{attribute 'qualified_only'}
{attribute 'global_init_slot' := '50500'}
VAR_GLOBAL PERSISTENT
	//These tags are created here because you cannot write directly to local scoped tags(cpt_3144) from outside the POU
	//They are created here then mapped to the local variables in the POU
	//All tags in this GVL MUST have the {attribute 'OPC.UA.DA' :='1'} string above them in order to be exposed to OPC
	//Tags that are ONLY being read from the HMI have their values set in the opc_mapping program
	
	//------------------------------------------------------------------------------------------------------------------


	//---System date time year-----------------------------------------------------------------------------------------------
	{attribute 'OPC.UA.DA' :='1'}
	popa_0082_system_date_time_year : INT;
	//System date time month
	{attribute 'OPC.UA.DA' :='1'}
	popa_0082_system_date_time_month : INT;
	//System date time day
	{attribute 'OPC.UA.DA' :='1'}
	popa_0082_system_date_time_day : INT;
	//System date time hour
	{attribute 'OPC.UA.DA' :='1'}
	popa_0082_system_date_time_hour : INT;
	//System date time minute
	{attribute 'OPC.UA.DA' :='1'}
	popa_0082_system_date_time_minute : INT;
	//System date time second
	{attribute 'OPC.UA.DA' :='1'}
	popa_0082_system_date_time_second : INT;
	//Hour setpoint for daily reset triggers
	{attribute 'OPC.UA.DA' :='1'}
	popa_0082_daily_reset_hour_setpoint : INT;
	//Minute setpoint for daily reset triggers
	{attribute 'OPC.UA.DA' :='1'}
	popa_0082_daily_reset_minute_setpoint : INT;
	//Alarm acknowledge, acks all alarms, clears lower priority level alarms
	{attribute 'OPC.UA.DA' :='1'}
	popa_0082_alarm_ack : BOOL;
	//Alarm reset, clears higher priority alarms
	{attribute 'OPC.UA.DA' :='1'}
	popa_0082_alarm_reset : BOOL;
	
//----------------------------------------------------------------------------------------------------------------------------------------		
	//State Mode
	{attribute 'OPC.UA.DA' :='1'}
	popa_0082_ed_routine_maint : BOOL;
	{attribute 'OPC.UA.DA' :='1'}
	popa_0082_ed_routine_idle : BOOL;
	{attribute 'OPC.UA.DA' :='1'}
	popa_0082_ed_routine_cip : BOOL;
	{attribute 'OPC.UA.DA' :='1'}
	popa_0082_ed_routine_stop : BOOL;
	{attribute 'OPC.UA.DA' :='1'}
	popa_0082_ed_routine_critical_stop : BOOL;
	
	
	//Safety
	{attribute 'OPC.UA.DA' :='1'}
	popa_0082_ed_safety_reset : BOOL;
	
	
//---HMI Commands--------------------------------------------------------------------------------------------------------------------------------------

	//Setpoints------------------------------------------------------------------------------------------------------------------
	{attribute 'OPC.UA.DA' :='1'}
	popa_0082_idle_pressure_setpoint_request : REAL;
	{attribute 'OPC.UA.DA' :='1'}
	popa_0082_cip_pressure_setpoint_request : REAL;
	{attribute 'OPC.UA.DA' :='1'}
	popa_0082_av_3148_b_hmi_position_request : REAL;
	{attribute 'OPC.UA.DA' :='1'}
	popa_0082_av_3248_b_hmi_position_request : REAL;
	{attribute 'OPC.UA.DA' :='1'}
	popa_0082_av_3348_b_hmi_position_request : REAL;
	
	//Pumps-----------------------------------------------------------------------------------------------------------------------
	{attribute 'OPC.UA.DA' :='1'}
	popa_0082_u_3112_b_hmi_start_request: BOOL;
	{attribute 'OPC.UA.DA' :='1'}
	popa_0082_u_3212_b_hmi_start_request: BOOL;
	{attribute 'OPC.UA.DA' :='1'}
	popa_0082_u_3312_b_hmi_start_request: BOOL;
	{attribute 'OPC.UA.DA' :='1'}
	popa_0082_u_3160_b_hmi_start_request: BOOL;
	{attribute 'OPC.UA.DA' :='1'}
	popa_0082_u_3260_b_hmi_start_request: BOOL;
	{attribute 'OPC.UA.DA' :='1'}
	popa_0082_u_3360_b_hmi_start_request: BOOL;
	{attribute 'OPC.UA.DA' :='1'}
	popa_0082_u_3370_b_hmi_start_request: BOOL;
	{attribute 'OPC.UA.DA' :='1'}
	popa_0092_u_3405_b_hmi_start_request: BOOL;
		
	{attribute 'OPC.UA.DA' :='1'}
	popa_0082_u_3112_b_hmi_speed_request: REAL;
	{attribute 'OPC.UA.DA' :='1'}
	popa_0082_u_3212_b_hmi_speed_request: REAL;
	{attribute 'OPC.UA.DA' :='1'}
	popa_0082_u_3312_b_hmi_speed_request: REAL;
	{attribute 'OPC.UA.DA' :='1'}
	popa_0082_u_3160_b_hmi_speed_request: REAL;
	{attribute 'OPC.UA.DA' :='1'}
	popa_0082_u_3260_b_hmi_speed_request: REAL;
	{attribute 'OPC.UA.DA' :='1'}
	popa_0082_u_3360_b_hmi_speed_request: REAL;
	{attribute 'OPC.UA.DA' :='1'}
	popa_0082_u_3370_b_hmi_speed_request: REAL;
	{attribute 'OPC.UA.DA' :='1'}
	popa_0092_u_3405_b_hmi_speed_request: REAL;
	
	//Valves------------------------------------------------------------------------------------------------------------------------------
	{attribute 'OPC.UA.DA' :='1'}
	popa_0082_nv_3110_b_hmi_open_request: BOOL;
	{attribute 'OPC.UA.DA' :='1'}
	popa_0082_nv_3210_b_hmi_open_request: BOOL;
	{attribute 'OPC.UA.DA' :='1'}
	popa_0082_nv_3310_b_hmi_open_request: BOOL;
	{attribute 'OPC.UA.DA' :='1'}
	popa_0082_nv_3135_b_hmi_open_request: BOOL;
	{attribute 'OPC.UA.DA' :='1'}
	popa_0082_nv_3235_b_hmi_open_request: BOOL;
	{attribute 'OPC.UA.DA' :='1'}
	popa_0082_nv_3335_b_hmi_open_request: BOOL;
	{attribute 'OPC.UA.DA' :='1'}
	popa_0082_nv_3372_b_hmi_open_request: BOOL;
	{attribute 'OPC.UA.DA' :='1'}
	popa_0082_nv_3162_b_hmi_open_request: BOOL;
	

	//-------------------------------------------------------------------------------------------
	//Digital valve open request
	{attribute 'OPC.UA.DA' :='1'}
	popa_0082_nv_3110_b_open_request : BOOL;
	//Digital valve status
	{attribute 'OPC.UA.DA' :='1'}
	popa_0082_nv_3110_b_status : INT;
	
	//Digital valve open request
	{attribute 'OPC.UA.DA' :='1'}
	popa_0082_nv_3210_b_open_request : BOOL;
	//Digital valve status
	{attribute 'OPC.UA.DA' :='1'}
	popa_0082_nv_3210_b_status : INT;
	
	//Digital valve open request
	{attribute 'OPC.UA.DA' :='1'}
	popa_0082_nv_3310_b_open_request : BOOL;
	//Digital valve status
	{attribute 'OPC.UA.DA' :='1'}
	popa_0082_nv_3310_b_status : INT;
	
	//Digital valve open request
	{attribute 'OPC.UA.DA' :='1'}
	popa_0082_nv_3135_b_open_request : BOOL;
	//Digital valve status
	{attribute 'OPC.UA.DA' :='1'}
	popa_0082_nv_3135_b_status : INT;
	
	//Digital valve open request
	{attribute 'OPC.UA.DA' :='1'}
	popa_0082_nv_3235_b_open_request : BOOL;
	//Digital valve status
	{attribute 'OPC.UA.DA' :='1'}
	popa_0082_nv_3235_b_status : INT;
	
	//Digital valve open request
	{attribute 'OPC.UA.DA' :='1'}
	popa_0082_nv_3335_b_open_request : BOOL;
	//Digital valve status
	{attribute 'OPC.UA.DA' :='1'}
	popa_0082_nv_3335_b_status : INT;
	
	//Digital valve open request
	{attribute 'OPC.UA.DA' :='1'}
	popa_0082_nv_3372_b_open_request : BOOL;
	//Digital valve status
	{attribute 'OPC.UA.DA' :='1'}
	popa_0082_nv_3372_b_status : INT;
	
	//Digital valve open request
	{attribute 'OPC.UA.DA' :='1'}
	popa_0082_nv_3162_b_open_request : BOOL;
	//Digital valve status
	{attribute 'OPC.UA.DA' :='1'}
	popa_0082_nv_3162_b_status : INT;
	
	//------------------------------------------------------------------------------------------------------------------
	//Alarm Priority setpoint
	{attribute 'OPC.UA.DA' :='1'}
	popa_0082_av_3148_b_position_fail_priority : INT;
	//Alarm delay setpoint(seconds)
	{attribute 'OPC.UA.DA' :='1'}
	popa_0082_av_3148_b_position_fail_delay_setpoint : INT;
	//Alarm active for HMI
	{attribute 'OPC.UA.DA' :='1'}
	popa_0082_av_3148_b_position_fail_active : BOOL;
	//Alarm enable
	{attribute 'OPC.UA.DA' :='1'}
	popa_0082_av_3148_b_position_fail_enable: BOOL;
	//------------------------------------------------------------------------------------------------------------------
	//Alarm Priority setpoint
	{attribute 'OPC.UA.DA' :='1'}
	popa_0082_av_3248_b_position_fail_priority : INT;
	//Alarm delay setpoint(seconds)
	{attribute 'OPC.UA.DA' :='1'}
	popa_0082_av_3248_b_position_fail_delay_setpoint : INT;
	//Alarm active for HMI
	{attribute 'OPC.UA.DA' :='1'}
	popa_0082_av_3248_b_position_fail_active : BOOL;
	//Alarm enable
	{attribute 'OPC.UA.DA' :='1'}
	popa_0082_av_3248_b_position_fail_enable: BOOL;
	//------------------------------------------------------------------------------------------------------------------
	//Alarm Priority setpoint
	{attribute 'OPC.UA.DA' :='1'}
	popa_0082_av_3348_b_position_fail_priority : INT;
	//Alarm delay setpoint(seconds)
	{attribute 'OPC.UA.DA' :='1'}
	popa_0082_av_3348_b_position_fail_delay_setpoint : INT;
	//Alarm active for HMI
	{attribute 'OPC.UA.DA' :='1'}
	popa_0082_av_3348_b_position_fail_active : BOOL;
	//Alarm enable
	{attribute 'OPC.UA.DA' :='1'}
	popa_0082_av_3348_b_position_fail_enable: BOOL;
	
	//------------------------------------------------------------------------------------------------------------------
	//Alarm Priority setpoint
	{attribute 'OPC.UA.DA' :='1'}
	popa_0082_nv_3110_b_fail_to_open_priority : INT;
	//Alarm delay setpoint(seconds)
	{attribute 'OPC.UA.DA' :='1'}
	popa_0082_nv_3110_b_fail_to_open_delay_setpoint : INT;
	//Alarm active for HMI
	{attribute 'OPC.UA.DA' :='1'}
	popa_0082_nv_3110_b_fail_to_open_active : BOOL;
	//Alarm enable
	{attribute 'OPC.UA.DA' :='1'}
	popa_0082_nv_3110_b_fail_to_open_enable: BOOL;
	
	//Alarm Priority setpoint
	{attribute 'OPC.UA.DA' :='1'}
	popa_0082_nv_3110_b_fail_to_close_priority : INT;
	//Alarm delay setpoint(seconds)
	{attribute 'OPC.UA.DA' :='1'}
	popa_0082_nv_3110_b_fail_to_close_delay_setpoint : INT;
	//Alarm active for HMI
	{attribute 'OPC.UA.DA' :='1'}
	popa_0082_nv_3110_b_fail_to_close_active : BOOL;
	//Alarm enable
	{attribute 'OPC.UA.DA' :='1'}
	popa_0082_nv_3110_b_fail_to_close_enable: BOOL;
	
	//------------------------------------------------------------------------------------------------------------------
	//Alarm Priority setpoint
	{attribute 'OPC.UA.DA' :='1'}
	popa_0082_nv_3210_b_fail_to_open_priority : INT;
	//Alarm delay setpoint(seconds)
	{attribute 'OPC.UA.DA' :='1'}
	popa_0082_nv_3210_b_fail_to_open_delay_setpoint : INT;
	//Alarm active for HMI
	{attribute 'OPC.UA.DA' :='1'}
	popa_0082_nv_3210_b_fail_to_open_active : BOOL;
	//Alarm enable
	{attribute 'OPC.UA.DA' :='1'}
	popa_0082_nv_3210_b_fail_to_open_enable: BOOL;
	
	//Alarm Priority setpoint
	{attribute 'OPC.UA.DA' :='1'}
	popa_0082_nv_3210_b_fail_to_close_priority : INT;
	//Alarm delay setpoint(seconds)
	{attribute 'OPC.UA.DA' :='1'}
	popa_0082_nv_3210_b_fail_to_close_delay_setpoint : INT;
	//Alarm active for HMI
	{attribute 'OPC.UA.DA' :='1'}
	popa_0082_nv_3210_b_fail_to_close_active : BOOL;
	//Alarm enable
	{attribute 'OPC.UA.DA' :='1'}
	popa_0082_nv_3210_b_fail_to_close_enable: BOOL;
	
	//------------------------------------------------------------------------------------------------------------------
	//Alarm Priority setpoint
	{attribute 'OPC.UA.DA' :='1'}
	popa_0082_nv_3310_b_fail_to_open_priority : INT;
	//Alarm delay setpoint(seconds)
	{attribute 'OPC.UA.DA' :='1'}
	popa_0082_nv_3310_b_fail_to_open_delay_setpoint : INT;
	//Alarm active for HMI
	{attribute 'OPC.UA.DA' :='1'}
	popa_0082_nv_3310_b_fail_to_open_active : BOOL;
	//Alarm enable
	{attribute 'OPC.UA.DA' :='1'}
	popa_0082_nv_3310_b_fail_to_open_enable: BOOL;
	
	//Alarm Priority setpoint
	{attribute 'OPC.UA.DA' :='1'}
	popa_0082_nv_3310_b_fail_to_close_priority : INT;
	//Alarm delay setpoint(seconds)
	{attribute 'OPC.UA.DA' :='1'}
	popa_0082_nv_3310_b_fail_to_close_delay_setpoint : INT;
	//Alarm active for HMI
	{attribute 'OPC.UA.DA' :='1'}
	popa_0082_nv_3310_b_fail_to_close_active : BOOL;
	//Alarm enable
	{attribute 'OPC.UA.DA' :='1'}
	popa_0082_nv_3310_b_fail_to_close_enable: BOOL;
	
	//------------------------------------------------------------------------------------------------------------------
	//Alarm Priority setpoint
	{attribute 'OPC.UA.DA' :='1'}
	popa_0082_nv_3135_b_fail_to_open_priority : INT;
	//Alarm delay setpoint(seconds)
	{attribute 'OPC.UA.DA' :='1'}
	popa_0082_nv_3135_b_fail_to_open_delay_setpoint : INT;
	//Alarm active for HMI
	{attribute 'OPC.UA.DA' :='1'}
	popa_0082_nv_3135_b_fail_to_open_active : BOOL;
	//Alarm enable
	{attribute 'OPC.UA.DA' :='1'}
	popa_0082_nv_3135_b_fail_to_open_enable: BOOL;
	
	//Alarm Priority setpoint
	{attribute 'OPC.UA.DA' :='1'}
	popa_0082_nv_3135_b_fail_to_close_priority : INT;
	//Alarm delay setpoint(seconds)
	{attribute 'OPC.UA.DA' :='1'}
	popa_0082_nv_3135_b_fail_to_close_delay_setpoint : INT;
	//Alarm active for HMI
	{attribute 'OPC.UA.DA' :='1'}
	popa_0082_nv_3135_b_fail_to_close_active : BOOL;
	//Alarm enable
	{attribute 'OPC.UA.DA' :='1'}
	popa_0082_nv_3135_b_fail_to_close_enable: BOOL;
	
	//------------------------------------------------------------------------------------------------------------------
	//Alarm Priority setpoint
	{attribute 'OPC.UA.DA' :='1'}
	popa_0082_nv_3235_b_fail_to_open_priority : INT;
	//Alarm delay setpoint(seconds)
	{attribute 'OPC.UA.DA' :='1'}
	popa_0082_nv_3235_b_fail_to_open_delay_setpoint : INT;
	//Alarm active for HMI
	{attribute 'OPC.UA.DA' :='1'}
	popa_0082_nv_3235_b_fail_to_open_active : BOOL;
	//Alarm enable
	{attribute 'OPC.UA.DA' :='1'}
	popa_0082_nv_3235_b_fail_to_open_enable: BOOL;
	
	//Alarm Priority setpoint
	{attribute 'OPC.UA.DA' :='1'}
	popa_0082_nv_3235_b_fail_to_close_priority : INT;
	//Alarm delay setpoint(seconds)
	{attribute 'OPC.UA.DA' :='1'}
	popa_0082_nv_3235_b_fail_to_close_delay_setpoint : INT;
	//Alarm active for HMI
	{attribute 'OPC.UA.DA' :='1'}
	popa_0082_nv_3235_b_fail_to_close_active : BOOL;
	//Alarm enable
	{attribute 'OPC.UA.DA' :='1'}
	popa_0082_nv_3235_b_fail_to_close_enable: BOOL;
	
	//------------------------------------------------------------------------------------------------------------------
	//Alarm Priority setpoint
	{attribute 'OPC.UA.DA' :='1'}
	popa_0082_nv_3335_b_fail_to_open_priority : INT;
	//Alarm delay setpoint(seconds)
	{attribute 'OPC.UA.DA' :='1'}
	popa_0082_nv_3335_b_fail_to_open_delay_setpoint : INT;
	//Alarm active for HMI
	{attribute 'OPC.UA.DA' :='1'}
	popa_0082_nv_3335_b_fail_to_open_active : BOOL;
	//Alarm enable
	{attribute 'OPC.UA.DA' :='1'}
	popa_0082_nv_3335_b_fail_to_open_enable: BOOL;
	
	//Alarm Priority setpoint
	{attribute 'OPC.UA.DA' :='1'}
	popa_0082_nv_3335_b_fail_to_close_priority : INT;
	//Alarm delay setpoint(seconds)
	{attribute 'OPC.UA.DA' :='1'}
	popa_0082_nv_3335_b_fail_to_close_delay_setpoint : INT;
	//Alarm active for HMI
	{attribute 'OPC.UA.DA' :='1'}
	popa_0082_nv_3335_b_fail_to_close_active : BOOL;
	//Alarm enable
	{attribute 'OPC.UA.DA' :='1'}
	popa_0082_nv_3335_b_fail_to_close_enable: BOOL;
	
	//------------------------------------------------------------------------------------------------------------------
	//Alarm Priority setpoint
	{attribute 'OPC.UA.DA' :='1'}
	popa_0082_nv_3372_b_fail_to_open_priority : INT;
	//Alarm delay setpoint(seconds)
	{attribute 'OPC.UA.DA' :='1'}
	popa_0082_nv_3372_b_fail_to_open_delay_setpoint : INT;
	//Alarm active for HMI
	{attribute 'OPC.UA.DA' :='1'}
	popa_0082_nv_3372_b_fail_to_open_active : BOOL;
	//Alarm enable
	{attribute 'OPC.UA.DA' :='1'}
	popa_0082_nv_3372_b_fail_to_open_enable: BOOL;
	
	//Alarm Priority setpoint
	{attribute 'OPC.UA.DA' :='1'}
	popa_0082_nv_3372_b_fail_to_close_priority : INT;
	//Alarm delay setpoint(seconds)
	{attribute 'OPC.UA.DA' :='1'}
	popa_0082_nv_3372_b_fail_to_close_delay_setpoint : INT;
	//Alarm active for HMI
	{attribute 'OPC.UA.DA' :='1'}
	popa_0082_nv_3372_b_fail_to_close_active : BOOL;
	//Alarm enable
	{attribute 'OPC.UA.DA' :='1'}
	popa_0082_nv_3372_b_fail_to_close_enable: BOOL;
	
	//------------------------------------------------------------------------------------------------------------------
	//Alarm Priority setpoint
	{attribute 'OPC.UA.DA' :='1'}
	popa_0082_nv_3162_b_fail_to_open_priority : INT;
	//Alarm delay setpoint(seconds)
	{attribute 'OPC.UA.DA' :='1'}
	popa_0082_nv_3162_b_fail_to_open_delay_setpoint : INT;
	//Alarm active for HMI
	{attribute 'OPC.UA.DA' :='1'}
	popa_0082_nv_3162_b_fail_to_open_active : BOOL;
	//Alarm enable
	{attribute 'OPC.UA.DA' :='1'}
	popa_0082_nv_3162_b_fail_to_open_enable: BOOL;
	
	//Alarm Priority setpoint
	{attribute 'OPC.UA.DA' :='1'}
	popa_0082_nv_3162_b_fail_to_close_priority : INT;
	//Alarm delay setpoint(seconds)
	{attribute 'OPC.UA.DA' :='1'}
	popa_0082_nv_3162_b_fail_to_close_delay_setpoint : INT;
	//Alarm active for HMI
	{attribute 'OPC.UA.DA' :='1'}
	popa_0082_nv_3162_b_fail_to_close_active : BOOL;
	//Alarm enable
	{attribute 'OPC.UA.DA' :='1'}
	popa_0082_nv_3162_b_fail_to_close_enable: BOOL;
	


//---Pumps-------------------------------------------------------------------------------------------------------------------------------------
	//------------------------------------------------------------------------------------------------------------------
	//Alarm Priority setpoint
	{attribute 'OPC.UA.DA' :='1'}
	popa_0082_u_3112_b_fail_to_start_priority : INT;
	//Alarm delay setpoint(seconds)
	{attribute 'OPC.UA.DA' :='1'}
	popa_0082_u_3112_b_fail_to_start_delay_setpoint : INT;
	//Alarm active for HMI
	{attribute 'OPC.UA.DA' :='1'}
	popa_0082_u_3112_b_fail_to_start_active : BOOL;
	//Alarm enable
	{attribute 'OPC.UA.DA' :='1'}
	popa_0082_u_3112_b_fail_to_start_enable: BOOL;
	
	//Alarm Priority setpoint
	{attribute 'OPC.UA.DA' :='1'}
	popa_0082_u_3112_b_fail_to_stop_priority : INT;
	//Alarm delay setpoint(seconds)
	{attribute 'OPC.UA.DA' :='1'}
	popa_0082_u_3112_b_fail_to_stop_delay_setpoint : INT;
	//Alarm active for HMI
	{attribute 'OPC.UA.DA' :='1'}
	popa_0082_u_3112_b_fail_to_stop_active : BOOL;
	//Alarm enable
	{attribute 'OPC.UA.DA' :='1'}
	popa_0082_u_3112_b_fail_to_stop_enable: BOOL;
	
	//------------------------------------------------------------------------------------------------------------------
	//Alarm Priority setpoint
	{attribute 'OPC.UA.DA' :='1'}
	popa_0082_u_3212_b_fail_to_start_priority : INT;
	//Alarm delay setpoint(seconds)
	{attribute 'OPC.UA.DA' :='1'}
	popa_0082_u_3212_b_fail_to_start_delay_setpoint : INT;
	//Alarm active for HMI
	{attribute 'OPC.UA.DA' :='1'}
	popa_0082_u_3212_b_fail_to_start_active : BOOL;
	//Alarm enable
	{attribute 'OPC.UA.DA' :='1'}
	popa_0082_u_3212_b_fail_to_start_enable: BOOL;
	
	//Alarm Priority setpoint
	{attribute 'OPC.UA.DA' :='1'}
	popa_0082_u_3212_b_fail_to_stop_priority : INT;
	//Alarm delay setpoint(seconds)
	{attribute 'OPC.UA.DA' :='1'}
	popa_0082_u_3212_b_fail_to_stop_delay_setpoint : INT;
	//Alarm active for HMI
	{attribute 'OPC.UA.DA' :='1'}
	popa_0082_u_3212_b_fail_to_stop_active : BOOL;
	//Alarm enable
	{attribute 'OPC.UA.DA' :='1'}
	popa_0082_u_3212_b_fail_to_stop_enable: BOOL;
	
	//------------------------------------------------------------------------------------------------------------------
	//Alarm Priority setpoint
	{attribute 'OPC.UA.DA' :='1'}
	popa_0082_u_3312_b_fail_to_start_priority : INT;
	//Alarm delay setpoint(seconds)
	{attribute 'OPC.UA.DA' :='1'}
	popa_0082_u_3312_b_fail_to_start_delay_setpoint : INT;
	//Alarm active for HMI
	{attribute 'OPC.UA.DA' :='1'}
	popa_0082_u_3312_b_fail_to_start_active : BOOL;
	//Alarm enable
	{attribute 'OPC.UA.DA' :='1'}
	popa_0082_u_3312_b_fail_to_start_enable: BOOL;
	
	//Alarm Priority setpoint
	{attribute 'OPC.UA.DA' :='1'}
	popa_0082_u_3312_b_fail_to_stop_priority : INT;
	//Alarm delay setpoint(seconds)
	{attribute 'OPC.UA.DA' :='1'}
	popa_0082_u_3312_b_fail_to_stop_delay_setpoint : INT;
	//Alarm active for HMI
	{attribute 'OPC.UA.DA' :='1'}
	popa_0082_u_3312_b_fail_to_stop_active : BOOL;
	//Alarm enable
	{attribute 'OPC.UA.DA' :='1'}
	popa_0082_u_3312_b_fail_to_stop_enable: BOOL;
	
	//------------------------------------------------------------------------------------------------------------------
	//Alarm Priority setpoint
	{attribute 'OPC.UA.DA' :='1'}
	popa_0082_u_3160_b_fail_to_start_priority : INT;
	//Alarm delay setpoint(seconds)
	{attribute 'OPC.UA.DA' :='1'}
	popa_0082_u_3160_b_fail_to_start_delay_setpoint : INT;
	//Alarm active for HMI
	{attribute 'OPC.UA.DA' :='1'}
	popa_0082_u_3160_b_fail_to_start_active : BOOL;
	//Alarm enable
	{attribute 'OPC.UA.DA' :='1'}
	popa_0082_u_3160_b_fail_to_start_enable: BOOL;
	
	//Alarm Priority setpoint
	{attribute 'OPC.UA.DA' :='1'}
	popa_0082_u_3160_b_fail_to_stop_priority : INT;
	//Alarm delay setpoint(seconds)
	{attribute 'OPC.UA.DA' :='1'}
	popa_0082_u_3160_b_fail_to_stop_delay_setpoint : INT;
	//Alarm active for HMI
	{attribute 'OPC.UA.DA' :='1'}
	popa_0082_u_3160_b_fail_to_stop_active : BOOL;
	//Alarm enable
	{attribute 'OPC.UA.DA' :='1'}
	popa_0082_u_3160_b_fail_to_stop_enable: BOOL;
	
	//------------------------------------------------------------------------------------------------------------------
	//Alarm Priority setpoint
	{attribute 'OPC.UA.DA' :='1'}
	popa_0082_u_3260_b_fail_to_start_priority : INT;
	//Alarm delay setpoint(seconds)
	{attribute 'OPC.UA.DA' :='1'}
	popa_0082_u_3260_b_fail_to_start_delay_setpoint : INT;
	//Alarm active for HMI
	{attribute 'OPC.UA.DA' :='1'}
	popa_0082_u_3260_b_fail_to_start_active : BOOL;
	//Alarm enable
	{attribute 'OPC.UA.DA' :='1'}
	popa_0082_u_3260_b_fail_to_start_enable: BOOL;
	
	//Alarm Priority setpoint
	{attribute 'OPC.UA.DA' :='1'}
	popa_0082_u_3260_b_fail_to_stop_priority : INT;
	//Alarm delay setpoint(seconds)
	{attribute 'OPC.UA.DA' :='1'}
	popa_0082_u_3260_b_fail_to_stop_delay_setpoint : INT;
	//Alarm active for HMI
	{attribute 'OPC.UA.DA' :='1'}
	popa_0082_u_3260_b_fail_to_stop_active : BOOL;
	//Alarm enable
	{attribute 'OPC.UA.DA' :='1'}
	popa_0082_u_3260_b_fail_to_stop_enable: BOOL;
	
	//------------------------------------------------------------------------------------------------------------------
	//Alarm Priority setpoint
	{attribute 'OPC.UA.DA' :='1'}
	popa_0082_u_3360_b_fail_to_start_priority : INT;
	//Alarm delay setpoint(seconds)
	{attribute 'OPC.UA.DA' :='1'}
	popa_0082_u_3360_b_fail_to_start_delay_setpoint : INT;
	//Alarm active for HMI
	{attribute 'OPC.UA.DA' :='1'}
	popa_0082_u_3360_b_fail_to_start_active : BOOL;
	//Alarm enable
	{attribute 'OPC.UA.DA' :='1'}
	popa_0082_u_3360_b_fail_to_start_enable: BOOL;
	
	//Alarm Priority setpoint
	{attribute 'OPC.UA.DA' :='1'}
	popa_0082_u_3360_b_fail_to_stop_priority : INT;
	//Alarm delay setpoint(seconds)
	{attribute 'OPC.UA.DA' :='1'}
	popa_0082_u_3360_b_fail_to_stop_delay_setpoint : INT;
	//Alarm active for HMI
	{attribute 'OPC.UA.DA' :='1'}
	popa_0082_u_3360_b_fail_to_stop_active : BOOL;
	//Alarm enable
	{attribute 'OPC.UA.DA' :='1'}
	popa_0082_u_3360_b_fail_to_stop_enable: BOOL;
	
	//------------------------------------------------------------------------------------------------------------------
	//Alarm Priority setpoint
	{attribute 'OPC.UA.DA' :='1'}
	popa_0082_u_3370_b_fail_to_start_priority : INT;
	//Alarm delay setpoint(seconds)
	{attribute 'OPC.UA.DA' :='1'}
	popa_0082_u_3370_b_fail_to_start_delay_setpoint : INT;
	//Alarm active for HMI
	{attribute 'OPC.UA.DA' :='1'}
	popa_0082_u_3370_b_fail_to_start_active : BOOL;
	//Alarm enable
	{attribute 'OPC.UA.DA' :='1'}
	popa_0082_u_3370_b_fail_to_start_enable: BOOL;
	
	//Alarm Priority setpoint
	{attribute 'OPC.UA.DA' :='1'}
	popa_0082_u_3370_b_fail_to_stop_priority : INT;
	//Alarm delay setpoint(seconds)
	{attribute 'OPC.UA.DA' :='1'}
	popa_0082_u_3370_b_fail_to_stop_delay_setpoint : INT;
	//Alarm active for HMI
	{attribute 'OPC.UA.DA' :='1'}
	popa_0082_u_3370_b_fail_to_stop_active : BOOL;
	//Alarm enable
	{attribute 'OPC.UA.DA' :='1'}
	popa_0082_u_3370_b_fail_to_stop_enable: BOOL;
	
	//------------------------------------------------------------------------------------------------------------------
	//Alarm Priority setpoint
	{attribute 'OPC.UA.DA' :='1'}
	popa_0092_u_3405_b_fail_to_start_priority : INT;
	//Alarm delay setpoint(seconds)
	{attribute 'OPC.UA.DA' :='1'}
	popa_0092_u_3405_b_fail_to_start_delay_setpoint : INT;
	//Alarm active for HMI
	{attribute 'OPC.UA.DA' :='1'}
	popa_0092_u_3405_b_fail_to_start_active : BOOL;
	//Alarm enable
	{attribute 'OPC.UA.DA' :='1'}
	popa_0092_u_3405_b_fail_to_start_enable: BOOL;
	
	//Alarm Priority setpoint
	{attribute 'OPC.UA.DA' :='1'}
	popa_0092_u_3405_b_fail_to_stop_priority : INT;
	//Alarm delay setpoint(seconds)
	{attribute 'OPC.UA.DA' :='1'}
	popa_0092_u_3405_b_fail_to_stop_delay_setpoint : INT;
	//Alarm active for HMI
	{attribute 'OPC.UA.DA' :='1'}
	popa_0092_u_3405_b_fail_to_stop_active : BOOL;
	//Alarm enable
	{attribute 'OPC.UA.DA' :='1'}
	popa_0092_u_3405_b_fail_to_stop_enable: BOOL;

	
	//---------------------------------------------------------------------------------------------------------
	//Raw Min value for analog input
	{attribute 'OPC.UA.DA' :='1'}
	popa_0082_u_3112_b_speed_command_raw_min : REAL :=0;
	//Raw max value for analog input
	{attribute 'OPC.UA.DA' :='1'}
	popa_0082_u_3112_b_speed_command_raw_max : REAL :=32767;
	//EU Min value for analog input
	{attribute 'OPC.UA.DA' :='1'}
	popa_0082_u_3112_b_speed_command_eu_min : REAL;
	//EU Max value for analog input
	{attribute 'OPC.UA.DA' :='1'}
	popa_0082_u_3112_b_speed_command_eu_max : REAL;
	//Filter factor value for analog input
	{attribute 'OPC.UA.DA' :='1'}
	popa_0082_u_3112_b_speed_command_filter_factor : REAL;
	//Scaled value for analog input
	{attribute 'OPC.UA.DA' :='1'}
	popa_0082_u_3112_b_speed_command_scaled_value : REAL;
	
	//Raw Min value for analog input
	{attribute 'OPC.UA.DA' :='1'}
	popa_0082_u_3112_b_speed_feedback_raw_min : REAL :=0;
	//Raw max value for analog input
	{attribute 'OPC.UA.DA' :='1'}
	popa_0082_u_3112_b_speed_feedback_raw_max : REAL :=32767;
	//EU Min value for analog input
	{attribute 'OPC.UA.DA' :='1'}
	popa_0082_u_3112_b_speed_feedback_eu_min : REAL;
	//EU Max value for analog input
	{attribute 'OPC.UA.DA' :='1'}
	popa_0082_u_3112_b_speed_feedback_eu_max : REAL;
	//Filter factor value for analog input
	{attribute 'OPC.UA.DA' :='1'}
	popa_0082_u_3112_b_speed_feedback_filter_factor : REAL;
	//Scaled value for analog input
	{attribute 'OPC.UA.DA' :='1'}
	popa_0082_u_3112_b_speed_feedback_scaled_value : REAL;
	
	
	//---------------------------------------------------------------------------------------------------------
	//Raw Min value for analog input
	{attribute 'OPC.UA.DA' :='1'}
	popa_0082_u_3212_b_speed_command_raw_min : REAL :=0;
	//Raw max value for analog input
	{attribute 'OPC.UA.DA' :='1'}
	popa_0082_u_3212_b_speed_command_raw_max : REAL :=32767;
	//EU Min value for analog input
	{attribute 'OPC.UA.DA' :='1'}
	popa_0082_u_3212_b_speed_command_eu_min : REAL;
	//EU Max value for analog input
	{attribute 'OPC.UA.DA' :='1'}
	popa_0082_u_3212_b_speed_command_eu_max : REAL;
	//Filter factor value for analog input
	{attribute 'OPC.UA.DA' :='1'}
	popa_0082_u_3212_b_speed_command_filter_factor : REAL;
	//Scaled value for analog input
	{attribute 'OPC.UA.DA' :='1'}
	popa_0082_u_3212_b_speed_command_scaled_value : REAL;
	
	//Raw Min value for analog input
	{attribute 'OPC.UA.DA' :='1'}
	popa_0082_u_3212_b_speed_feedback_raw_min : REAL :=0;
	//Raw max value for analog input
	{attribute 'OPC.UA.DA' :='1'}
	popa_0082_u_3212_b_speed_feedback_raw_max : REAL :=32767;
	//EU Min value for analog input
	{attribute 'OPC.UA.DA' :='1'}
	popa_0082_u_3212_b_speed_feedback_eu_min : REAL;
	//EU Max value for analog input
	{attribute 'OPC.UA.DA' :='1'}
	popa_0082_u_3212_b_speed_feedback_eu_max : REAL;
	//Filter factor value for analog input
	{attribute 'OPC.UA.DA' :='1'}
	popa_0082_u_3212_b_speed_feedback_filter_factor : REAL;
	//Scaled value for analog input
	{attribute 'OPC.UA.DA' :='1'}
	popa_0082_u_3212_b_speed_feedback_scaled_value : REAL;
	
	
	//---------------------------------------------------------------------------------------------------------
	//Raw Min value for analog input
	{attribute 'OPC.UA.DA' :='1'}
	popa_0082_u_3312_b_speed_command_raw_min : REAL :=0;
	//Raw max value for analog input
	{attribute 'OPC.UA.DA' :='1'}
	popa_0082_u_3312_b_speed_command_raw_max : REAL :=32767;
	//EU Min value for analog input
	{attribute 'OPC.UA.DA' :='1'}
	popa_0082_u_3312_b_speed_command_eu_min : REAL;
	//EU Max value for analog input
	{attribute 'OPC.UA.DA' :='1'}
	popa_0082_u_3312_b_speed_command_eu_max : REAL;
	//Filter factor value for analog input
	{attribute 'OPC.UA.DA' :='1'}
	popa_0082_u_3312_b_speed_command_filter_factor : REAL;
	//Scaled value for analog input
	{attribute 'OPC.UA.DA' :='1'}
	popa_0082_u_3312_b_speed_command_scaled_value : REAL;
	
	//Raw Min value for analog input
	{attribute 'OPC.UA.DA' :='1'}
	popa_0082_u_3312_b_speed_feedback_raw_min : REAL :=0;
	//Raw max value for analog input
	{attribute 'OPC.UA.DA' :='1'}
	popa_0082_u_3312_b_speed_feedback_raw_max : REAL :=32767;
	//EU Min value for analog input
	{attribute 'OPC.UA.DA' :='1'}
	popa_0082_u_3312_b_speed_feedback_eu_min : REAL;
	//EU Max value for analog input
	{attribute 'OPC.UA.DA' :='1'}
	popa_0082_u_3312_b_speed_feedback_eu_max : REAL;
	//Filter factor value for analog input
	{attribute 'OPC.UA.DA' :='1'}
	popa_0082_u_3312_b_speed_feedback_filter_factor : REAL;
	//Scaled value for analog input
	{attribute 'OPC.UA.DA' :='1'}
	popa_0082_u_3312_b_speed_feedback_scaled_value : REAL;
	
	
	//---------------------------------------------------------------------------------------------------------
	//Raw Min value for analog input
	{attribute 'OPC.UA.DA' :='1'}
	popa_0082_u_3160_b_speed_command_raw_min : REAL :=0;
	//Raw max value for analog input
	{attribute 'OPC.UA.DA' :='1'}
	popa_0082_u_3160_b_speed_command_raw_max : REAL :=32767;
	//EU Min value for analog input
	{attribute 'OPC.UA.DA' :='1'}
	popa_0082_u_3160_b_speed_command_eu_min : REAL;
	//EU Max value for analog input
	{attribute 'OPC.UA.DA' :='1'}
	popa_0082_u_3160_b_speed_command_eu_max : REAL;
	//Filter factor value for analog input
	{attribute 'OPC.UA.DA' :='1'}
	popa_0082_u_3160_b_speed_command_filter_factor : REAL;
	//Scaled value for analog input
	{attribute 'OPC.UA.DA' :='1'}
	popa_0082_u_3160_b_speed_command_scaled_value : REAL;
	
	//Raw Min value for analog input
	{attribute 'OPC.UA.DA' :='1'}
	popa_0082_u_3160_b_speed_feedback_raw_min : REAL :=0;
	//Raw max value for analog input
	{attribute 'OPC.UA.DA' :='1'}
	popa_0082_u_3160_b_speed_feedback_raw_max : REAL :=32767;
	//EU Min value for analog input
	{attribute 'OPC.UA.DA' :='1'}
	popa_0082_u_3160_b_speed_feedback_eu_min : REAL;
	//EU Max value for analog input
	{attribute 'OPC.UA.DA' :='1'}
	popa_0082_u_3160_b_speed_feedback_eu_max : REAL;
	//Filter factor value for analog input
	{attribute 'OPC.UA.DA' :='1'}
	popa_0082_u_3160_b_speed_feedback_filter_factor : REAL;
	//Scaled value for analog input
	{attribute 'OPC.UA.DA' :='1'}
	popa_0082_u_3160_b_speed_feedback_scaled_value : REAL;
	
	
	//---------------------------------------------------------------------------------------------------------
	//Raw Min value for analog input
	{attribute 'OPC.UA.DA' :='1'}
	popa_0082_u_3260_b_speed_command_raw_min : REAL :=0;
	//Raw max value for analog input
	{attribute 'OPC.UA.DA' :='1'}
	popa_0082_u_3260_b_speed_command_raw_max : REAL :=32767;
	//EU Min value for analog input
	{attribute 'OPC.UA.DA' :='1'}
	popa_0082_u_3260_b_speed_command_eu_min : REAL;
	//EU Max value for analog input
	{attribute 'OPC.UA.DA' :='1'}
	popa_0082_u_3260_b_speed_command_eu_max : REAL;
	//Filter factor value for analog input
	{attribute 'OPC.UA.DA' :='1'}
	popa_0082_u_3260_b_speed_command_filter_factor : REAL;
	//Scaled value for analog input
	{attribute 'OPC.UA.DA' :='1'}
	popa_0082_u_3260_b_speed_command_scaled_value : REAL;
	
	//Raw Min value for analog input
	{attribute 'OPC.UA.DA' :='1'}
	popa_0082_u_3260_b_speed_feedback_raw_min : REAL :=0;
	//Raw max value for analog input
	{attribute 'OPC.UA.DA' :='1'}
	popa_0082_u_3260_b_speed_feedback_raw_max : REAL :=32767;
	//EU Min value for analog input
	{attribute 'OPC.UA.DA' :='1'}
	popa_0082_u_3260_b_speed_feedback_eu_min : REAL;
	//EU Max value for analog input
	{attribute 'OPC.UA.DA' :='1'}
	popa_0082_u_3260_b_speed_feedback_eu_max : REAL;
	//Filter factor value for analog input
	{attribute 'OPC.UA.DA' :='1'}
	popa_0082_u_3260_b_speed_feedback_filter_factor : REAL;
	//Scaled value for analog input
	{attribute 'OPC.UA.DA' :='1'}
	popa_0082_u_3260_b_speed_feedback_scaled_value : REAL;
	
	
	//---------------------------------------------------------------------------------------------------------
	//Raw Min value for analog input
	{attribute 'OPC.UA.DA' :='1'}
	popa_0082_u_3360_b_speed_command_raw_min : REAL :=0;
	//Raw max value for analog input
	{attribute 'OPC.UA.DA' :='1'}
	popa_0082_u_3360_b_speed_command_raw_max : REAL :=32767;
	//EU Min value for analog input
	{attribute 'OPC.UA.DA' :='1'}
	popa_0082_u_3360_b_speed_command_eu_min : REAL;
	//EU Max value for analog input
	{attribute 'OPC.UA.DA' :='1'}
	popa_0082_u_3360_b_speed_command_eu_max : REAL;
	//Filter factor value for analog input
	{attribute 'OPC.UA.DA' :='1'}
	popa_0082_u_3360_b_speed_command_filter_factor : REAL;
	//Scaled value for analog input
	{attribute 'OPC.UA.DA' :='1'}
	popa_0082_u_3360_b_speed_command_scaled_value : REAL;
	
	//Raw Min value for analog input
	{attribute 'OPC.UA.DA' :='1'}
	popa_0082_u_3360_b_speed_feedback_raw_min : REAL :=0;
	//Raw max value for analog input
	{attribute 'OPC.UA.DA' :='1'}
	popa_0082_u_3360_b_speed_feedback_raw_max : REAL :=32767;
	//EU Min value for analog input
	{attribute 'OPC.UA.DA' :='1'}
	popa_0082_u_3360_b_speed_feedback_eu_min : REAL;
	//EU Max value for analog input
	{attribute 'OPC.UA.DA' :='1'}
	popa_0082_u_3360_b_speed_feedback_eu_max : REAL;
	//Filter factor value for analog input
	{attribute 'OPC.UA.DA' :='1'}
	popa_0082_u_3360_b_speed_feedback_filter_factor : REAL;
	//Scaled value for analog input
	{attribute 'OPC.UA.DA' :='1'}
	popa_0082_u_3360_b_speed_feedback_scaled_value : REAL;
	
	
	//---------------------------------------------------------------------------------------------------------
	//Raw Min value for analog input
	{attribute 'OPC.UA.DA' :='1'}
	popa_0082_u_3370_b_speed_command_raw_min : REAL :=0;
	//Raw max value for analog input
	{attribute 'OPC.UA.DA' :='1'}
	popa_0082_u_3370_b_speed_command_raw_max : REAL :=32767;
	//EU Min value for analog input
	{attribute 'OPC.UA.DA' :='1'}
	popa_0082_u_3370_b_speed_command_eu_min : REAL;
	//EU Max value for analog input
	{attribute 'OPC.UA.DA' :='1'}
	popa_0082_u_3370_b_speed_command_eu_max : REAL;
	//Filter factor value for analog input
	{attribute 'OPC.UA.DA' :='1'}
	popa_0082_u_3370_b_speed_command_filter_factor : REAL;
	//Scaled value for analog input
	{attribute 'OPC.UA.DA' :='1'}
	popa_0082_u_3370_b_speed_command_scaled_value : REAL;
	
	//Raw Min value for analog input
	{attribute 'OPC.UA.DA' :='1'}
	popa_0082_u_3370_b_speed_feedback_raw_min : REAL :=0;
	//Raw max value for analog input
	{attribute 'OPC.UA.DA' :='1'}
	popa_0082_u_3370_b_speed_feedback_raw_max : REAL :=32767;
	//EU Min value for analog input
	{attribute 'OPC.UA.DA' :='1'}
	popa_0082_u_3370_b_speed_feedback_eu_min : REAL;
	//EU Max value for analog input
	{attribute 'OPC.UA.DA' :='1'}
	popa_0082_u_3370_b_speed_feedback_eu_max : REAL;
	//Filter factor value for analog input
	{attribute 'OPC.UA.DA' :='1'}
	popa_0082_u_3370_b_speed_feedback_filter_factor : REAL;
	//Scaled value for analog input
	{attribute 'OPC.UA.DA' :='1'}
	popa_0082_u_3370_b_speed_feedback_scaled_value : REAL;
	
	
	//---------------------------------------------------------------------------------------------------------
	//Raw Min value for analog input
	{attribute 'OPC.UA.DA' :='1'}
	popa_0092_u_3405_b_speed_command_raw_min : REAL :=0;
	//Raw max value for analog input
	{attribute 'OPC.UA.DA' :='1'}
	popa_0092_u_3405_b_speed_command_raw_max : REAL :=32767;
	//EU Min value for analog input
	{attribute 'OPC.UA.DA' :='1'}
	popa_0092_u_3405_b_speed_command_eu_min : REAL;
	//EU Max value for analog input
	{attribute 'OPC.UA.DA' :='1'}
	popa_0092_u_3405_b_speed_command_eu_max : REAL;
	//Filter factor value for analog input
	{attribute 'OPC.UA.DA' :='1'}
	popa_0092_u_3405_b_speed_command_filter_factor : REAL;
	//Scaled value for analog input
	{attribute 'OPC.UA.DA' :='1'}
	popa_0092_u_3405_b_speed_command_scaled_value : REAL;
	
	//Raw Min value for analog input
	{attribute 'OPC.UA.DA' :='1'}
	popa_0092_u_3405_b_speed_feedback_raw_min : REAL :=0;
	//Raw max value for analog input
	{attribute 'OPC.UA.DA' :='1'}
	popa_0092_u_3405_b_speed_feedback_raw_max : REAL :=32767;
	//EU Min value for analog input
	{attribute 'OPC.UA.DA' :='1'}
	popa_0092_u_3405_b_speed_feedback_eu_min : REAL;
	//EU Max value for analog input
	{attribute 'OPC.UA.DA' :='1'}
	popa_0092_u_3405_b_speed_feedback_eu_max : REAL;
	//Filter factor value for analog input
	{attribute 'OPC.UA.DA' :='1'}
	popa_0092_u_3405_b_speed_feedback_filter_factor : REAL;
	//Scaled value for analog input
	{attribute 'OPC.UA.DA' :='1'}
	popa_0092_u_3405_b_speed_feedback_scaled_value : REAL;
	
//---Valves----------------------------------------------------------------------------------------------------------------------------------------

	//Raw Min value for analog input
	{attribute 'OPC.UA.DA' :='1'}
	popa_0082_av_3148_b_position_feedback_raw_min : REAL :=0;
	//Raw max value for analog input
	{attribute 'OPC.UA.DA' :='1'}
	popa_0082_av_3148_b_position_feedback_raw_max : REAL :=32767;
	//EU Min value for analog input
	{attribute 'OPC.UA.DA' :='1'}
	popa_0082_av_3148_b_position_feedback_eu_min : REAL;
	//EU Max value for analog input
	{attribute 'OPC.UA.DA' :='1'}
	popa_0082_av_3148_b_position_feedback_eu_max : REAL;
	//Filter factor value for analog input
	{attribute 'OPC.UA.DA' :='1'}
	popa_0082_av_3148_b_position_feedback_filter_factor : REAL;
	//Scaled value for analog input
	{attribute 'OPC.UA.DA' :='1'}
	popa_0082_av_3148_b_position_feedback_scaled_value : REAL;
	
	//Raw Min value for analog input
	{attribute 'OPC.UA.DA' :='1'}
	popa_0082_av_3148_b_position_command_raw_min : REAL :=0;
	//Raw max value for analog input
	{attribute 'OPC.UA.DA' :='1'}
	popa_0082_av_3148_b_position_command_raw_max : REAL :=32767;
	//EU Min value for analog input
	{attribute 'OPC.UA.DA' :='1'}
	popa_0082_av_3148_b_position_command_eu_min : REAL;
	//EU Max value for analog input
	{attribute 'OPC.UA.DA' :='1'}
	popa_0082_av_3148_b_position_command_eu_max : REAL;
	//Filter factor value for analog input
	{attribute 'OPC.UA.DA' :='1'}
	popa_0082_av_3148_b_position_command_filter_factor : REAL;
	//Scaled value for analog input
	{attribute 'OPC.UA.DA' :='1'}
	popa_0082_av_3148_b_position_command_scaled_value : REAL;
//-----------------------------------------------------------------------------------------------------------	
	//Raw Min value for analog input
	{attribute 'OPC.UA.DA' :='1'}
	popa_0082_av_3248_b_position_feedback_raw_min : REAL :=0;
	//Raw max value for analog input
	{attribute 'OPC.UA.DA' :='1'}
	popa_0082_av_3248_b_position_feedback_raw_max : REAL :=32767;
	//EU Min value for analog input
	{attribute 'OPC.UA.DA' :='1'}
	popa_0082_av_3248_b_position_feedback_eu_min : REAL;
	//EU Max value for analog input
	{attribute 'OPC.UA.DA' :='1'}
	popa_0082_av_3248_b_position_feedback_eu_max : REAL;
	//Filter factor value for analog input
	{attribute 'OPC.UA.DA' :='1'}
	popa_0082_av_3248_b_position_feedback_filter_factor : REAL;
	//Scaled value for analog input
	{attribute 'OPC.UA.DA' :='1'}
	popa_0082_av_3248_b_position_feedback_scaled_value : REAL;
	
	//Raw Min value for analog input
	{attribute 'OPC.UA.DA' :='1'}
	popa_0082_av_3248_b_position_command_raw_min : REAL :=0;
	//Raw max value for analog input
	{attribute 'OPC.UA.DA' :='1'}
	popa_0082_av_3248_b_position_command_raw_max : REAL :=32767;
	//EU Min value for analog input
	{attribute 'OPC.UA.DA' :='1'}
	popa_0082_av_3248_b_position_command_eu_min : REAL;
	//EU Max value for analog input
	{attribute 'OPC.UA.DA' :='1'}
	popa_0082_av_3248_b_position_command_eu_max : REAL;
	//Filter factor value for analog input
	{attribute 'OPC.UA.DA' :='1'}
	popa_0082_av_3248_b_position_command_filter_factor : REAL;
	//Scaled value for analog input
	{attribute 'OPC.UA.DA' :='1'}
	popa_0082_av_3248_b_position_command_scaled_value : REAL;
//-----------------------------------------------------------------------------------------------------------	

	//Raw Min value for analog input
	{attribute 'OPC.UA.DA' :='1'}
	popa_0082_av_3348_b_position_feedback_raw_min : REAL :=0;
	//Raw max value for analog input
	{attribute 'OPC.UA.DA' :='1'}
	popa_0082_av_3348_b_position_feedback_raw_max : REAL :=32767;
	//EU Min value for analog input
	{attribute 'OPC.UA.DA' :='1'}
	popa_0082_av_3348_b_position_feedback_eu_min : REAL;
	//EU Max value for analog input
	{attribute 'OPC.UA.DA' :='1'}
	popa_0082_av_3348_b_position_feedback_eu_max : REAL;
	//Filter factor value for analog input
	{attribute 'OPC.UA.DA' :='1'}
	popa_0082_av_3348_b_position_feedback_filter_factor : REAL;
	//Scaled value for analog input
	{attribute 'OPC.UA.DA' :='1'}
	popa_0082_av_3348_b_position_feedback_scaled_value : REAL;
	
	//Raw Min value for analog input
	{attribute 'OPC.UA.DA' :='1'}
	popa_0082_av_3348_b_position_command_raw_min : REAL :=0;
	//Raw max value for analog input
	{attribute 'OPC.UA.DA' :='1'}
	popa_0082_av_3348_b_position_command_raw_max : REAL :=32767;
	//EU Min value for analog input
	{attribute 'OPC.UA.DA' :='1'}
	popa_0082_av_3348_b_position_command_eu_min : REAL;
	//EU Max value for analog input
	{attribute 'OPC.UA.DA' :='1'}
	popa_0082_av_3348_b_position_command_eu_max : REAL;
	//Filter factor value for analog input
	{attribute 'OPC.UA.DA' :='1'}
	popa_0082_av_3348_b_position_command_filter_factor : REAL;
	//Scaled value for analog input
	{attribute 'OPC.UA.DA' :='1'}
	popa_0082_av_3348_b_position_command_scaled_value : REAL;
//-----------------------------------------------------------------------------------------------------------		


	//Example motor starter runtime maintenance reset
	{attribute 'OPC.UA.DA' :='1'}
	popa_0082_u_3160_b_runtime_maint_reset : BOOL;
	//Example motor starter run request
	{attribute 'OPC.UA.DA' :='1'}
	popa_0082_u_3160_b_run_request : BOOL;
	//Example motor starter runtime today
	{attribute 'OPC.UA.DA' :='1'}
	popa_0082_u_3160_b_runtime_today : REAL;
	//Example motor starter runtime total
	{attribute 'OPC.UA.DA' :='1'}
	popa_0082_u_3160_b_runtime_total : REAL;
	//Example motor starter runtime maint
	{attribute 'OPC.UA.DA' :='1'}
	popa_0082_u_3160_b_runtime_maint : REAL;
	//Example motor starter status, 0=Off, 1=Run, 2=Fault
	{attribute 'OPC.UA.DA' :='1'}
	popa_0082_u_3160_b_status : REAL;
	
	//--------------------------------------------------------------------------------------------------------------
	//Example motor vfd runtime maintenance reset
	{attribute 'OPC.UA.DA' :='1'}
	popa_0082_u_3112_b_runtime_maint_reset : BOOL;
	//Example motor vfd run request
	{attribute 'OPC.UA.DA' :='1'}
	popa_0082_u_3112_b_run_request : BOOL;
	//Example motor vfd speed request
	{attribute 'OPC.UA.DA' :='1'}
	popa_0082_u_3112_b_speed_request : REAL;
	//Example motor vfd speed feedback
	{attribute 'OPC.UA.DA' :='1'}
	popa_0082_u_3112_b_speed_feedback : REAL;
	//Example motor vfd runtime today
	{attribute 'OPC.UA.DA' :='1'}
	popa_0082_u_3112_b_runtime_today : REAL;
	//Example motor vfd runtime total
	{attribute 'OPC.UA.DA' :='1'}
	popa_0082_u_3112_b_runtime_total : REAL;
	//Example motor vfd runtime maint
	{attribute 'OPC.UA.DA' :='1'}
	popa_0082_u_3112_b_runtime_maint : REAL;
	//Example motor vfd status, 0=Off, 1=Run, 2=Fault
	{attribute 'OPC.UA.DA' :='1'}
	popa_0082_u_3112_b_status : REAL;
	
	//--------------------------------------------------------------------------------------------------------------
	//Example motor vfd runtime maintenance reset
	{attribute 'OPC.UA.DA' :='1'}
	popa_0082_u_3212_b_runtime_maint_reset : BOOL;
	//Example motor vfd run request
	{attribute 'OPC.UA.DA' :='1'}
	popa_0082_u_3212_b_run_request : BOOL;
	//Example motor vfd speed request
	{attribute 'OPC.UA.DA' :='1'}
	popa_0082_u_3212_b_speed_request : REAL;
	//Example motor vfd speed feedback
	{attribute 'OPC.UA.DA' :='1'}
	popa_0082_u_3212_b_speed_feedback : REAL;
	//Example motor vfd runtime today
	{attribute 'OPC.UA.DA' :='1'}
	popa_0082_u_3212_b_runtime_today : REAL;
	//Example motor vfd runtime total
	{attribute 'OPC.UA.DA' :='1'}
	popa_0082_u_3212_b_runtime_total : REAL;
	//Example motor vfd runtime maint
	{attribute 'OPC.UA.DA' :='1'}
	popa_0082_u_3212_b_runtime_maint : REAL;
	//Example motor vfd status, 0=Off, 1=Run, 2=Fault
	{attribute 'OPC.UA.DA' :='1'}
	popa_0082_u_3212_b_status : REAL;
	
	//--------------------------------------------------------------------------------------------------------------
	//Example motor vfd runtime maintenance reset
	{attribute 'OPC.UA.DA' :='1'}
	popa_0082_u_3312_b_runtime_maint_reset : BOOL;
	//Example motor vfd run request
	{attribute 'OPC.UA.DA' :='1'}
	popa_0082_u_3312_b_run_request : BOOL;
	//Example motor vfd speed request
	{attribute 'OPC.UA.DA' :='1'}
	popa_0082_u_3312_b_speed_request : REAL;
	//Example motor vfd speed feedback
	{attribute 'OPC.UA.DA' :='1'}
	popa_0082_u_3312_b_speed_feedback : REAL;
	//Example motor vfd runtime today
	{attribute 'OPC.UA.DA' :='1'}
	popa_0082_u_3312_b_runtime_today : REAL;
	//Example motor vfd runtime total
	{attribute 'OPC.UA.DA' :='1'}
	popa_0082_u_3312_b_runtime_total : REAL;
	//Example motor vfd runtime maint
	{attribute 'OPC.UA.DA' :='1'}
	popa_0082_u_3312_b_runtime_maint : REAL;
	//Example motor vfd status, 0=Off, 1=Run, 2=Fault
	{attribute 'OPC.UA.DA' :='1'}
	popa_0082_u_3312_b_status : REAL;
	
	//--------------------------------------------------------------------------------------------------------------
	
	//Example motor vfd speed request
	{attribute 'OPC.UA.DA' :='1'}
	popa_0082_u_3160_b_speed_request : REAL;
	//Example motor vfd speed feedback
	{attribute 'OPC.UA.DA' :='1'}
	popa_0082_u_3160_b_speed_feedback : REAL;

	
	
	//--------------------------------------------------------------------------------------------------------------
	//Example motor vfd runtime maintenance reset
	{attribute 'OPC.UA.DA' :='1'}
	popa_0082_u_3260_b_runtime_maint_reset : BOOL;
	//Example motor vfd run request
	{attribute 'OPC.UA.DA' :='1'}
	popa_0082_u_3260_b_run_request : BOOL;
	//Example motor vfd speed request
	{attribute 'OPC.UA.DA' :='1'}
	popa_0082_u_3260_b_speed_request : REAL;
	//Example motor vfd speed feedback
	{attribute 'OPC.UA.DA' :='1'}
	popa_0082_u_3260_b_speed_feedback : REAL;
	//Example motor vfd runtime today
	{attribute 'OPC.UA.DA' :='1'}
	popa_0082_u_3260_b_runtime_today : REAL;
	//Example motor vfd runtime total
	{attribute 'OPC.UA.DA' :='1'}
	popa_0082_u_3260_b_runtime_total : REAL;
	//Example motor vfd runtime maint
	{attribute 'OPC.UA.DA' :='1'}
	popa_0082_u_3260_b_runtime_maint : REAL;
	//Example motor vfd status, 0=Off, 1=Run, 2=Fault
	{attribute 'OPC.UA.DA' :='1'}
	popa_0082_u_3260_b_status : REAL;
	
	//--------------------------------------------------------------------------------------------------------------
	//Example motor vfd runtime maintenance reset
	{attribute 'OPC.UA.DA' :='1'}
	popa_0082_u_3360_b_runtime_maint_reset : BOOL;
	//Example motor vfd run request
	{attribute 'OPC.UA.DA' :='1'}
	popa_0082_u_3360_b_run_request : BOOL;
	//Example motor vfd speed request
	{attribute 'OPC.UA.DA' :='1'}
	popa_0082_u_3360_b_speed_request : REAL;
	//Example motor vfd speed feedback
	{attribute 'OPC.UA.DA' :='1'}
	popa_0082_u_3360_b_speed_feedback : REAL;
	//Example motor vfd runtime today
	{attribute 'OPC.UA.DA' :='1'}
	popa_0082_u_3360_b_runtime_today : REAL;
	//Example motor vfd runtime total
	{attribute 'OPC.UA.DA' :='1'}
	popa_0082_u_3360_b_runtime_total : REAL;
	//Example motor vfd runtime maint
	{attribute 'OPC.UA.DA' :='1'}
	popa_0082_u_3360_b_runtime_maint : REAL;
	//Example motor vfd status, 0=Off, 1=Run, 2=Fault
	{attribute 'OPC.UA.DA' :='1'}
	popa_0082_u_3360_b_status : REAL;
	
	//--------------------------------------------------------------------------------------------------------------
	//Example motor vfd runtime maintenance reset
	{attribute 'OPC.UA.DA' :='1'}
	popa_0082_u_3370_b_runtime_maint_reset : BOOL;
	//Example motor vfd run request
	{attribute 'OPC.UA.DA' :='1'}
	popa_0082_u_3370_b_run_request : BOOL;
	//Example motor vfd speed request
	{attribute 'OPC.UA.DA' :='1'}
	popa_0082_u_3370_b_speed_request : REAL;
	//Example motor vfd speed feedback
	{attribute 'OPC.UA.DA' :='1'}
	popa_0082_u_3370_b_speed_feedback : REAL;
	//Example motor vfd runtime today
	{attribute 'OPC.UA.DA' :='1'}
	popa_0082_u_3370_b_runtime_today : REAL;
	//Example motor vfd runtime total
	{attribute 'OPC.UA.DA' :='1'}
	popa_0082_u_3370_b_runtime_total : REAL;
	//Example motor vfd runtime maint
	{attribute 'OPC.UA.DA' :='1'}
	popa_0082_u_3370_b_runtime_maint : REAL;
	//Example motor vfd status, 0=Off, 1=Run, 2=Fault
	{attribute 'OPC.UA.DA' :='1'}
	popa_0082_u_3370_b_status : REAL;
	
	//--------------------------------------------------------------------------------------------------------------
	//Example motor vfd runtime maintenance reset
	{attribute 'OPC.UA.DA' :='1'}
	popa_0092_u_3405_b_runtime_maint_reset : BOOL;
	//Example motor vfd run request
	{attribute 'OPC.UA.DA' :='1'}
	popa_0092_u_3405_b_run_request : BOOL;
	//Example motor vfd speed request
	{attribute 'OPC.UA.DA' :='1'}
	popa_0092_u_3405_b_speed_request : REAL;
	//Example motor vfd speed feedback
	{attribute 'OPC.UA.DA' :='1'}
	popa_0092_u_3405_b_speed_feedback : REAL;
	//Example motor vfd runtime today
	{attribute 'OPC.UA.DA' :='1'}
	popa_0092_u_3405_b_runtime_today : REAL;
	//Example motor vfd runtime total
	{attribute 'OPC.UA.DA' :='1'}
	popa_0092_u_3405_b_runtime_total : REAL;
	//Example motor vfd runtime maint
	{attribute 'OPC.UA.DA' :='1'}
	popa_0092_u_3405_b_runtime_maint : REAL;
	//Example motor vfd status, 0=Off, 1=Run, 2=Fault
	{attribute 'OPC.UA.DA' :='1'}
	popa_0092_u_3405_b_status : REAL;
	
	
	//Analog valve position request
	{attribute 'OPC.UA.DA' :='1'}
	popa_0082_av_3148_b_position_feedback : REAL;
	//Example analog valve position request
	{attribute 'OPC.UA.DA' :='1'}
	popa_0082_av_3148_b_position_request : REAL;
	//Example analog valve position fail deadband
	{attribute 'OPC.UA.DA' :='1'}
	popa_0082_av_3148_b_position_deadband_sp : REAL;
	//Example analog valve position requested when in fault state
	{attribute 'OPC.UA.DA' :='1'}
	popa_0082_av_3148_b_position_faulted : REAL;
	//Example analog valve status
	{attribute 'OPC.UA.DA' :='1'}
	popa_0082_av_3148_b_status : INT;
	//-------------------------------------------------------------------------------------------
		{attribute 'OPC.UA.DA' :='1'}
	popa_0082_av_3248_b_position_feedback : REAL;
	//Example analog valve position request
	{attribute 'OPC.UA.DA' :='1'}
	popa_0082_av_3248_b_position_request : REAL;
	//Example analog valve position fail deadband
	{attribute 'OPC.UA.DA' :='1'}
	popa_0082_av_3248_b_position_deadband_sp : REAL;
	//Example analog valve position requested when in fault state
	{attribute 'OPC.UA.DA' :='1'}
	popa_0082_av_3248_b_position_faulted : REAL;
	//Example analog valve status
	{attribute 'OPC.UA.DA' :='1'}
	popa_0082_av_3248_b_status : INT;
	//-------------------------------------------------------------------------------------------
		{attribute 'OPC.UA.DA' :='1'}
	popa_0082_av_3348_b_position_feedback : REAL;
	//Example analog valve position request
	{attribute 'OPC.UA.DA' :='1'}
	popa_0082_av_3348_b_position_request : REAL;
	//Example analog valve position fail deadband
	{attribute 'OPC.UA.DA' :='1'}
	popa_0082_av_3348_b_position_deadband_sp : REAL;
	//Example analog valve position requested when in fault state
	{attribute 'OPC.UA.DA' :='1'}
	popa_0082_av_3348_b_position_faulted : REAL;
	//Example analog valve status
	{attribute 'OPC.UA.DA' :='1'}
	popa_0082_av_3348_b_status : INT;
	
	
	
	
//---Sensors----------------------------------------------------------------------------------------------------------------------------	
	//---cpt_3144-----------------------------------------------------------------------------------------------------------------------
	//Alarm Priority setpoint
	{attribute 'OPC.UA.DA' :='1'}
	popa_0082_cpt_3144_b_low_low_priority : INT;
	//Alarm delay setpoint(seconds)
	{attribute 'OPC.UA.DA' :='1'}
	popa_0082_cpt_3144_b_low_low_delay_setpoint : INT;
	//Alarm active for HMI
	{attribute 'OPC.UA.DA' :='1'}
	popa_0082_cpt_3144_b_low_low_active : BOOL;
	//Analog Alarm Setpoint
	{attribute 'OPC.UA.DA' :='1'}
	popa_0082_cpt_3144_b_low_low_setpoint : REAL;
	//Alarm enable
	{attribute 'OPC.UA.DA' :='1'}
	popa_0082_cpt_3144_b_low_low_enable: BOOL;
	
	//Alarm Priority setpoint
	{attribute 'OPC.UA.DA' :='1'}
	popa_0082_cpt_3144_b_low_priority : INT;
	//Alarm delay setpoint(seconds)
	{attribute 'OPC.UA.DA' :='1'}
	popa_0082_cpt_3144_b_low_delay_setpoint : INT;
	//Alarm active for HMI
	{attribute 'OPC.UA.DA' :='1'}
	popa_0082_cpt_3144_b_low_active : BOOL;
	//Analog Alarm Setpoint
	{attribute 'OPC.UA.DA' :='1'}
	popa_0082_cpt_3144_b_low_setpoint : REAL;
	//Alarm enable
	{attribute 'OPC.UA.DA' :='1'}
	popa_0082_cpt_3144_b_low_enable: BOOL;
	
	//Alarm Priority setpoint
	{attribute 'OPC.UA.DA' :='1'}
	popa_0082_cpt_3144_b_high_priority : INT;
	//Alarm delay setpoint(seconds)
	{attribute 'OPC.UA.DA' :='1'}
	popa_0082_cpt_3144_b_high_delay_setpoint : INT;
	//Alarm active for HMI
	{attribute 'OPC.UA.DA' :='1'}
	popa_0082_cpt_3144_b_high_active : BOOL;
	//Analog Alarm Setpoint
	{attribute 'OPC.UA.DA' :='1'}
	popa_0082_cpt_3144_b_high_setpoint : REAL;
	//Alarm enable
	{attribute 'OPC.UA.DA' :='1'}
	popa_0082_cpt_3144_b_high_enable: BOOL;
	
	//Alarm Priority setpoint
	{attribute 'OPC.UA.DA' :='1'}
	popa_0082_cpt_3144_b_high_high_priority : INT;
	//Alarm delay setpoint(seconds)
	{attribute 'OPC.UA.DA' :='1'}
	popa_0082_cpt_3144_b_high_high_delay_setpoint : INT;
	//Alarm active for HMI
	{attribute 'OPC.UA.DA' :='1'}
	popa_0082_cpt_3144_b_high_high_active : BOOL;
	//Analog Alarm Setpoint
	{attribute 'OPC.UA.DA' :='1'}
	popa_0082_cpt_3144_b_high_high_setpoint : REAL;
	//Alarm enable
	{attribute 'OPC.UA.DA' :='1'}
	popa_0082_cpt_3144_b_high_high_enable: BOOL;
	
	
	//Raw Min value for analog input
	{attribute 'OPC.UA.DA' :='1'}
	popa_0082_cpt_3144_b_raw_min : REAL :=0;
	//Raw max value for analog input
	{attribute 'OPC.UA.DA' :='1'}
	popa_0082_cpt_3144_b_raw_max : REAL :=32767;
	//EU Min value for analog input
	{attribute 'OPC.UA.DA' :='1'}
	popa_0082_cpt_3144_b_eu_min : REAL;
	//EU Max value for analog input
	{attribute 'OPC.UA.DA' :='1'}
	popa_0082_cpt_3144_b_eu_max : REAL;
	//Filter factor value for analog input
	{attribute 'OPC.UA.DA' :='1'}
	popa_0082_cpt_3144_b_filter_factor : REAL;
	//Scaled value for analog input
	{attribute 'OPC.UA.DA' :='1'}
	popa_0082_cpt_3144_b_scaled_value : REAL;
	
	//---cct_3120-----------------------------------------------------------------------------------------------------------------------
	//Alarm Priority setpoint
	{attribute 'OPC.UA.DA' :='1'}
	popa_0082_cct_3120_b_low_low_priority : INT;
	//Alarm delay setpoint(seconds)
	{attribute 'OPC.UA.DA' :='1'}
	popa_0082_cct_3120_b_low_low_delay_setpoint : INT;
	//Alarm active for HMI
	{attribute 'OPC.UA.DA' :='1'}
	popa_0082_cct_3120_b_low_low_active : BOOL;
	//Analog Alarm Setpoint
	{attribute 'OPC.UA.DA' :='1'}
	popa_0082_cct_3120_b_low_low_setpoint : REAL;
	//Alarm enable
	{attribute 'OPC.UA.DA' :='1'}
	popa_0082_cct_3120_b_low_low_enable: BOOL;
	
	//Alarm Priority setpoint
	{attribute 'OPC.UA.DA' :='1'}
	popa_0082_cct_3120_b_low_priority : INT;
	//Alarm delay setpoint(seconds)
	{attribute 'OPC.UA.DA' :='1'}
	popa_0082_cct_3120_b_low_delay_setpoint : INT;
	//Alarm active for HMI
	{attribute 'OPC.UA.DA' :='1'}
	popa_0082_cct_3120_b_low_active : BOOL;
	//Analog Alarm Setpoint
	{attribute 'OPC.UA.DA' :='1'}
	popa_0082_cct_3120_b_low_setpoint : REAL;
	//Alarm enable
	{attribute 'OPC.UA.DA' :='1'}
	popa_0082_cct_3120_b_low_enable: BOOL;
	
	//Alarm Priority setpoint
	{attribute 'OPC.UA.DA' :='1'}
	popa_0082_cct_3120_b_high_priority : INT;
	//Alarm delay setpoint(seconds)
	{attribute 'OPC.UA.DA' :='1'}
	popa_0082_cct_3120_b_high_delay_setpoint : INT;
	//Alarm active for HMI
	{attribute 'OPC.UA.DA' :='1'}
	popa_0082_cct_3120_b_high_active : BOOL;
	//Analog Alarm Setpoint
	{attribute 'OPC.UA.DA' :='1'}
	popa_0082_cct_3120_b_high_setpoint : REAL;
	//Alarm enable
	{attribute 'OPC.UA.DA' :='1'}
	popa_0082_cct_3120_b_high_enable: BOOL;
	
	//Alarm Priority setpoint
	{attribute 'OPC.UA.DA' :='1'}
	popa_0082_cct_3120_b_high_high_priority : INT;
	//Alarm delay setpoint(seconds)
	{attribute 'OPC.UA.DA' :='1'}
	popa_0082_cct_3120_b_high_high_delay_setpoint : INT;
	//Alarm active for HMI
	{attribute 'OPC.UA.DA' :='1'}
	popa_0082_cct_3120_b_high_high_active : BOOL;
	//Analog Alarm Setpoint
	{attribute 'OPC.UA.DA' :='1'}
	popa_0082_cct_3120_b_high_high_setpoint : REAL;
	//Alarm enable
	{attribute 'OPC.UA.DA' :='1'}
	popa_0082_cct_3120_b_high_high_enable: BOOL;
	
	
	//Raw Min value for analog input
	{attribute 'OPC.UA.DA' :='1'}
	popa_0082_cct_3120_b_raw_min : REAL :=0;
	//Raw max value for analog input
	{attribute 'OPC.UA.DA' :='1'}
	popa_0082_cct_3120_b_raw_max : REAL :=32767;
	//EU Min value for analog input
	{attribute 'OPC.UA.DA' :='1'}
	popa_0082_cct_3120_b_eu_min : REAL;
	//EU Max value for analog input
	{attribute 'OPC.UA.DA' :='1'}
	popa_0082_cct_3120_b_eu_max : REAL;
	//Filter factor value for analog input
	{attribute 'OPC.UA.DA' :='1'}
	popa_0082_cct_3120_b_filter_factor : REAL;
	//Scaled value for analog input
	{attribute 'OPC.UA.DA' :='1'}
	popa_0082_cct_3120_b_scaled_value : REAL;
	
		//---cct_3220-----------------------------------------------------------------------------------------------------------------------
	//Alarm Priority setpoint
	{attribute 'OPC.UA.DA' :='1'}
	popa_0082_cct_3220_b_low_low_priority : INT;
	//Alarm delay setpoint(seconds)
	{attribute 'OPC.UA.DA' :='1'}
	popa_0082_cct_3220_b_low_low_delay_setpoint : INT;
	//Alarm active for HMI
	{attribute 'OPC.UA.DA' :='1'}
	popa_0082_cct_3220_b_low_low_active : BOOL;
	//Analog Alarm Setpoint
	{attribute 'OPC.UA.DA' :='1'}
	popa_0082_cct_3220_b_low_low_setpoint : REAL;
	//Alarm enable
	{attribute 'OPC.UA.DA' :='1'}
	popa_0082_cct_3220_b_low_low_enable: BOOL;
	
	//Alarm Priority setpoint
	{attribute 'OPC.UA.DA' :='1'}
	popa_0082_cct_3220_b_low_priority : INT;
	//Alarm delay setpoint(seconds)
	{attribute 'OPC.UA.DA' :='1'}
	popa_0082_cct_3220_b_low_delay_setpoint : INT;
	//Alarm active for HMI
	{attribute 'OPC.UA.DA' :='1'}
	popa_0082_cct_3220_b_low_active : BOOL;
	//Analog Alarm Setpoint
	{attribute 'OPC.UA.DA' :='1'}
	popa_0082_cct_3220_b_low_setpoint : REAL;
	//Alarm enable
	{attribute 'OPC.UA.DA' :='1'}
	popa_0082_cct_3220_b_low_enable: BOOL;
	
	//Alarm Priority setpoint
	{attribute 'OPC.UA.DA' :='1'}
	popa_0082_cct_3220_b_high_priority : INT;
	//Alarm delay setpoint(seconds)
	{attribute 'OPC.UA.DA' :='1'}
	popa_0082_cct_3220_b_high_delay_setpoint : INT;
	//Alarm active for HMI
	{attribute 'OPC.UA.DA' :='1'}
	popa_0082_cct_3220_b_high_active : BOOL;
	//Analog Alarm Setpoint
	{attribute 'OPC.UA.DA' :='1'}
	popa_0082_cct_3220_b_high_setpoint : REAL;
	//Alarm enable
	{attribute 'OPC.UA.DA' :='1'}
	popa_0082_cct_3220_b_high_enable: BOOL;
	
	//Alarm Priority setpoint
	{attribute 'OPC.UA.DA' :='1'}
	popa_0082_cct_3220_b_high_high_priority : INT;
	//Alarm delay setpoint(seconds)
	{attribute 'OPC.UA.DA' :='1'}
	popa_0082_cct_3220_b_high_high_delay_setpoint : INT;
	//Alarm active for HMI
	{attribute 'OPC.UA.DA' :='1'}
	popa_0082_cct_3220_b_high_high_active : BOOL;
	//Analog Alarm Setpoint
	{attribute 'OPC.UA.DA' :='1'}
	popa_0082_cct_3220_b_high_high_setpoint : REAL;
	//Alarm enable
	{attribute 'OPC.UA.DA' :='1'}
	popa_0082_cct_3220_b_high_high_enable: BOOL;
	
	
	//Raw Min value for analog input
	{attribute 'OPC.UA.DA' :='1'}
	popa_0082_cct_3220_b_raw_min : REAL :=0;
	//Raw max value for analog input
	{attribute 'OPC.UA.DA' :='1'}
	popa_0082_cct_3220_b_raw_max : REAL :=32767;
	//EU Min value for analog input
	{attribute 'OPC.UA.DA' :='1'}
	popa_0082_cct_3220_b_eu_min : REAL;
	//EU Max value for analog input
	{attribute 'OPC.UA.DA' :='1'}
	popa_0082_cct_3220_b_eu_max : REAL;
	//Filter factor value for analog input
	{attribute 'OPC.UA.DA' :='1'}
	popa_0082_cct_3220_b_filter_factor : REAL;
	//Scaled value for analog input
	{attribute 'OPC.UA.DA' :='1'}
	popa_0082_cct_3220_b_scaled_value : REAL;
	
		//---cct_3320-----------------------------------------------------------------------------------------------------------------------
	//Alarm Priority setpoint
	{attribute 'OPC.UA.DA' :='1'}
	popa_0082_cct_3320_b_low_low_priority : INT;
	//Alarm delay setpoint(seconds)
	{attribute 'OPC.UA.DA' :='1'}
	popa_0082_cct_3320_b_low_low_delay_setpoint : INT;
	//Alarm active for HMI
	{attribute 'OPC.UA.DA' :='1'}
	popa_0082_cct_3320_b_low_low_active : BOOL;
	//Analog Alarm Setpoint
	{attribute 'OPC.UA.DA' :='1'}
	popa_0082_cct_3320_b_low_low_setpoint : REAL;
	//Alarm enable
	{attribute 'OPC.UA.DA' :='1'}
	popa_0082_cct_3320_b_low_low_enable: BOOL;
	
	//Alarm Priority setpoint
	{attribute 'OPC.UA.DA' :='1'}
	popa_0082_cct_3320_b_low_priority : INT;
	//Alarm delay setpoint(seconds)
	{attribute 'OPC.UA.DA' :='1'}
	popa_0082_cct_3320_b_low_delay_setpoint : INT;
	//Alarm active for HMI
	{attribute 'OPC.UA.DA' :='1'}
	popa_0082_cct_3320_b_low_active : BOOL;
	//Analog Alarm Setpoint
	{attribute 'OPC.UA.DA' :='1'}
	popa_0082_cct_3320_b_low_setpoint : REAL;
	//Alarm enable
	{attribute 'OPC.UA.DA' :='1'}
	popa_0082_cct_3320_b_low_enable: BOOL;
	
	//Alarm Priority setpoint
	{attribute 'OPC.UA.DA' :='1'}
	popa_0082_cct_3320_b_high_priority : INT;
	//Alarm delay setpoint(seconds)
	{attribute 'OPC.UA.DA' :='1'}
	popa_0082_cct_3320_b_high_delay_setpoint : INT;
	//Alarm active for HMI
	{attribute 'OPC.UA.DA' :='1'}
	popa_0082_cct_3320_b_high_active : BOOL;
	//Analog Alarm Setpoint
	{attribute 'OPC.UA.DA' :='1'}
	popa_0082_cct_3320_b_high_setpoint : REAL;
	//Alarm enable
	{attribute 'OPC.UA.DA' :='1'}
	popa_0082_cct_3320_b_high_enable: BOOL;
	
	//Alarm Priority setpoint
	{attribute 'OPC.UA.DA' :='1'}
	popa_0082_cct_3320_b_high_high_priority : INT;
	//Alarm delay setpoint(seconds)
	{attribute 'OPC.UA.DA' :='1'}
	popa_0082_cct_3320_b_high_high_delay_setpoint : INT;
	//Alarm active for HMI
	{attribute 'OPC.UA.DA' :='1'}
	popa_0082_cct_3320_b_high_high_active : BOOL;
	//Analog Alarm Setpoint
	{attribute 'OPC.UA.DA' :='1'}
	popa_0082_cct_3320_b_high_high_setpoint : REAL;
	//Alarm enable
	{attribute 'OPC.UA.DA' :='1'}
	popa_0082_cct_3320_b_high_high_enable: BOOL;
	
	
	//Raw Min value for analog input
	{attribute 'OPC.UA.DA' :='1'}
	popa_0082_cct_3320_b_raw_min : REAL :=0;
	//Raw max value for analog input
	{attribute 'OPC.UA.DA' :='1'}
	popa_0082_cct_3320_b_raw_max : REAL :=32767;
	//EU Min value for analog input
	{attribute 'OPC.UA.DA' :='1'}
	popa_0082_cct_3320_b_eu_min : REAL;
	//EU Max value for analog input
	{attribute 'OPC.UA.DA' :='1'}
	popa_0082_cct_3320_b_eu_max : REAL;
	//Filter factor value for analog input
	{attribute 'OPC.UA.DA' :='1'}
	popa_0082_cct_3320_b_filter_factor : REAL;
	//Scaled value for analog input
	{attribute 'OPC.UA.DA' :='1'}
	popa_0082_cct_3320_b_scaled_value : REAL;
	
		//---cct_3142-----------------------------------------------------------------------------------------------------------------------
	//Alarm Priority setpoint
	{attribute 'OPC.UA.DA' :='1'}
	popa_0082_cct_3142_b_low_low_priority : INT;
	//Alarm delay setpoint(seconds)
	{attribute 'OPC.UA.DA' :='1'}
	popa_0082_cct_3142_b_low_low_delay_setpoint : INT;
	//Alarm active for HMI
	{attribute 'OPC.UA.DA' :='1'}
	popa_0082_cct_3142_b_low_low_active : BOOL;
	//Analog Alarm Setpoint
	{attribute 'OPC.UA.DA' :='1'}
	popa_0082_cct_3142_b_low_low_setpoint : REAL;
	//Alarm enable
	{attribute 'OPC.UA.DA' :='1'}
	popa_0082_cct_3142_b_low_low_enable: BOOL;
	
	//Alarm Priority setpoint
	{attribute 'OPC.UA.DA' :='1'}
	popa_0082_cct_3142_b_low_priority : INT;
	//Alarm delay setpoint(seconds)
	{attribute 'OPC.UA.DA' :='1'}
	popa_0082_cct_3142_b_low_delay_setpoint : INT;
	//Alarm active for HMI
	{attribute 'OPC.UA.DA' :='1'}
	popa_0082_cct_3142_b_low_active : BOOL;
	//Analog Alarm Setpoint
	{attribute 'OPC.UA.DA' :='1'}
	popa_0082_cct_3142_b_low_setpoint : REAL;
	//Alarm enable
	{attribute 'OPC.UA.DA' :='1'}
	popa_0082_cct_3142_b_low_enable: BOOL;
	
	//Alarm Priority setpoint
	{attribute 'OPC.UA.DA' :='1'}
	popa_0082_cct_3142_b_high_priority : INT;
	//Alarm delay setpoint(seconds)
	{attribute 'OPC.UA.DA' :='1'}
	popa_0082_cct_3142_b_high_delay_setpoint : INT;
	//Alarm active for HMI
	{attribute 'OPC.UA.DA' :='1'}
	popa_0082_cct_3142_b_high_active : BOOL;
	//Analog Alarm Setpoint
	{attribute 'OPC.UA.DA' :='1'}
	popa_0082_cct_3142_b_high_setpoint : REAL;
	//Alarm enable
	{attribute 'OPC.UA.DA' :='1'}
	popa_0082_cct_3142_b_high_enable: BOOL;
	
	//Alarm Priority setpoint
	{attribute 'OPC.UA.DA' :='1'}
	popa_0082_cct_3142_b_high_high_priority : INT;
	//Alarm delay setpoint(seconds)
	{attribute 'OPC.UA.DA' :='1'}
	popa_0082_cct_3142_b_high_high_delay_setpoint : INT;
	//Alarm active for HMI
	{attribute 'OPC.UA.DA' :='1'}
	popa_0082_cct_3142_b_high_high_active : BOOL;
	//Analog Alarm Setpoint
	{attribute 'OPC.UA.DA' :='1'}
	popa_0082_cct_3142_b_high_high_setpoint : REAL;
	//Alarm enable
	{attribute 'OPC.UA.DA' :='1'}
	popa_0082_cct_3142_b_high_high_enable: BOOL;
	
	
	//Raw Min value for analog input
	{attribute 'OPC.UA.DA' :='1'}
	popa_0082_cct_3142_b_raw_min : REAL :=0;
	//Raw max value for analog input
	{attribute 'OPC.UA.DA' :='1'}
	popa_0082_cct_3142_b_raw_max : REAL :=32767;
	//EU Min value for analog input
	{attribute 'OPC.UA.DA' :='1'}
	popa_0082_cct_3142_b_eu_min : REAL;
	//EU Max value for analog input
	{attribute 'OPC.UA.DA' :='1'}
	popa_0082_cct_3142_b_eu_max : REAL;
	//Filter factor value for analog input
	{attribute 'OPC.UA.DA' :='1'}
	popa_0082_cct_3142_b_filter_factor : REAL;
	//Scaled value for analog input
	{attribute 'OPC.UA.DA' :='1'}
	popa_0082_cct_3142_b_scaled_value : REAL;
	
		//---cct_3242-----------------------------------------------------------------------------------------------------------------------
	//Alarm Priority setpoint
	{attribute 'OPC.UA.DA' :='1'}
	popa_0082_cct_3242_b_low_low_priority : INT;
	//Alarm delay setpoint(seconds)
	{attribute 'OPC.UA.DA' :='1'}
	popa_0082_cct_3242_b_low_low_delay_setpoint : INT;
	//Alarm active for HMI
	{attribute 'OPC.UA.DA' :='1'}
	popa_0082_cct_3242_b_low_low_active : BOOL;
	//Analog Alarm Setpoint
	{attribute 'OPC.UA.DA' :='1'}
	popa_0082_cct_3242_b_low_low_setpoint : REAL;
	//Alarm enable
	{attribute 'OPC.UA.DA' :='1'}
	popa_0082_cct_3242_b_low_low_enable: BOOL;
	
	//Alarm Priority setpoint
	{attribute 'OPC.UA.DA' :='1'}
	popa_0082_cct_3242_b_low_priority : INT;
	//Alarm delay setpoint(seconds)
	{attribute 'OPC.UA.DA' :='1'}
	popa_0082_cct_3242_b_low_delay_setpoint : INT;
	//Alarm active for HMI
	{attribute 'OPC.UA.DA' :='1'}
	popa_0082_cct_3242_b_low_active : BOOL;
	//Analog Alarm Setpoint
	{attribute 'OPC.UA.DA' :='1'}
	popa_0082_cct_3242_b_low_setpoint : REAL;
	//Alarm enable
	{attribute 'OPC.UA.DA' :='1'}
	popa_0082_cct_3242_b_low_enable: BOOL;
	
	//Alarm Priority setpoint
	{attribute 'OPC.UA.DA' :='1'}
	popa_0082_cct_3242_b_high_priority : INT;
	//Alarm delay setpoint(seconds)
	{attribute 'OPC.UA.DA' :='1'}
	popa_0082_cct_3242_b_high_delay_setpoint : INT;
	//Alarm active for HMI
	{attribute 'OPC.UA.DA' :='1'}
	popa_0082_cct_3242_b_high_active : BOOL;
	//Analog Alarm Setpoint
	{attribute 'OPC.UA.DA' :='1'}
	popa_0082_cct_3242_b_high_setpoint : REAL;
	//Alarm enable
	{attribute 'OPC.UA.DA' :='1'}
	popa_0082_cct_3242_b_high_enable: BOOL;
	
	//Alarm Priority setpoint
	{attribute 'OPC.UA.DA' :='1'}
	popa_0082_cct_3242_b_high_high_priority : INT;
	//Alarm delay setpoint(seconds)
	{attribute 'OPC.UA.DA' :='1'}
	popa_0082_cct_3242_b_high_high_delay_setpoint : INT;
	//Alarm active for HMI
	{attribute 'OPC.UA.DA' :='1'}
	popa_0082_cct_3242_b_high_high_active : BOOL;
	//Analog Alarm Setpoint
	{attribute 'OPC.UA.DA' :='1'}
	popa_0082_cct_3242_b_high_high_setpoint : REAL;
	//Alarm enable
	{attribute 'OPC.UA.DA' :='1'}
	popa_0082_cct_3242_b_high_high_enable: BOOL;
	
	
	//Raw Min value for analog input
	{attribute 'OPC.UA.DA' :='1'}
	popa_0082_cct_3242_b_raw_min : REAL :=0;
	//Raw max value for analog input
	{attribute 'OPC.UA.DA' :='1'}
	popa_0082_cct_3242_b_raw_max : REAL :=32767;
	//EU Min value for analog input
	{attribute 'OPC.UA.DA' :='1'}
	popa_0082_cct_3242_b_eu_min : REAL;
	//EU Max value for analog input
	{attribute 'OPC.UA.DA' :='1'}
	popa_0082_cct_3242_b_eu_max : REAL;
	//Filter factor value for analog input
	{attribute 'OPC.UA.DA' :='1'}
	popa_0082_cct_3242_b_filter_factor : REAL;
	//Scaled value for analog input
	{attribute 'OPC.UA.DA' :='1'}
	popa_0082_cct_3242_b_scaled_value : REAL;
	
		//---cct_3342-----------------------------------------------------------------------------------------------------------------------
	//Alarm Priority setpoint
	{attribute 'OPC.UA.DA' :='1'}
	popa_0082_cct_3342_b_low_low_priority : INT;
	//Alarm delay setpoint(seconds)
	{attribute 'OPC.UA.DA' :='1'}
	popa_0082_cct_3342_b_low_low_delay_setpoint : INT;
	//Alarm active for HMI
	{attribute 'OPC.UA.DA' :='1'}
	popa_0082_cct_3342_b_low_low_active : BOOL;
	//Analog Alarm Setpoint
	{attribute 'OPC.UA.DA' :='1'}
	popa_0082_cct_3342_b_low_low_setpoint : REAL;
	//Alarm enable
	{attribute 'OPC.UA.DA' :='1'}
	popa_0082_cct_3342_b_low_low_enable: BOOL;
	
	//Alarm Priority setpoint
	{attribute 'OPC.UA.DA' :='1'}
	popa_0082_cct_3342_b_low_priority : INT;
	//Alarm delay setpoint(seconds)
	{attribute 'OPC.UA.DA' :='1'}
	popa_0082_cct_3342_b_low_delay_setpoint : INT;
	//Alarm active for HMI
	{attribute 'OPC.UA.DA' :='1'}
	popa_0082_cct_3342_b_low_active : BOOL;
	//Analog Alarm Setpoint
	{attribute 'OPC.UA.DA' :='1'}
	popa_0082_cct_3342_b_low_setpoint : REAL;
	//Alarm enable
	{attribute 'OPC.UA.DA' :='1'}
	popa_0082_cct_3342_b_low_enable: BOOL;
	
	//Alarm Priority setpoint
	{attribute 'OPC.UA.DA' :='1'}
	popa_0082_cct_3342_b_high_priority : INT;
	//Alarm delay setpoint(seconds)
	{attribute 'OPC.UA.DA' :='1'}
	popa_0082_cct_3342_b_high_delay_setpoint : INT;
	//Alarm active for HMI
	{attribute 'OPC.UA.DA' :='1'}
	popa_0082_cct_3342_b_high_active : BOOL;
	//Analog Alarm Setpoint
	{attribute 'OPC.UA.DA' :='1'}
	popa_0082_cct_3342_b_high_setpoint : REAL;
	//Alarm enable
	{attribute 'OPC.UA.DA' :='1'}
	popa_0082_cct_3342_b_high_enable: BOOL;
	
	//Alarm Priority setpoint
	{attribute 'OPC.UA.DA' :='1'}
	popa_0082_cct_3342_b_high_high_priority : INT;
	//Alarm delay setpoint(seconds)
	{attribute 'OPC.UA.DA' :='1'}
	popa_0082_cct_3342_b_high_high_delay_setpoint : INT;
	//Alarm active for HMI
	{attribute 'OPC.UA.DA' :='1'}
	popa_0082_cct_3342_b_high_high_active : BOOL;
	//Analog Alarm Setpoint
	{attribute 'OPC.UA.DA' :='1'}
	popa_0082_cct_3342_b_high_high_setpoint : REAL;
	//Alarm enable
	{attribute 'OPC.UA.DA' :='1'}
	popa_0082_cct_3342_b_high_high_enable: BOOL;
	
	
	//Raw Min value for analog input
	{attribute 'OPC.UA.DA' :='1'}
	popa_0082_cct_3342_b_raw_min : REAL :=0;
	//Raw max value for analog input
	{attribute 'OPC.UA.DA' :='1'}
	popa_0082_cct_3342_b_raw_max : REAL :=32767;
	//EU Min value for analog input
	{attribute 'OPC.UA.DA' :='1'}
	popa_0082_cct_3342_b_eu_min : REAL;
	//EU Max value for analog input
	{attribute 'OPC.UA.DA' :='1'}
	popa_0082_cct_3342_b_eu_max : REAL;
	//Filter factor value for analog input
	{attribute 'OPC.UA.DA' :='1'}
	popa_0082_cct_3342_b_filter_factor : REAL;
	//Scaled value for analog input
	{attribute 'OPC.UA.DA' :='1'}
	popa_0082_cct_3342_b_scaled_value : REAL;

	//---ft_3122-----------------------------------------------------------------------------------------------------------------------
	//Alarm Priority setpoint
	{attribute 'OPC.UA.DA' :='1'}
	popa_0082_ft_3122_b_low_low_priority : INT;
	//Alarm delay setpoint(seconds)
	{attribute 'OPC.UA.DA' :='1'}
	popa_0082_ft_3122_b_low_low_delay_setpoint : INT;
	//Alarm active for HMI
	{attribute 'OPC.UA.DA' :='1'}
	popa_0082_ft_3122_b_low_low_active : BOOL;
	//Analog Alarm Setpoint
	{attribute 'OPC.UA.DA' :='1'}
	popa_0082_ft_3122_b_low_low_setpoint : REAL;
	//Alarm enable
	{attribute 'OPC.UA.DA' :='1'}
	popa_0082_ft_3122_b_low_low_enable: BOOL;
	
	//Alarm Priority setpoint
	{attribute 'OPC.UA.DA' :='1'}
	popa_0082_ft_3122_b_low_priority : INT;
	//Alarm delay setpoint(seconds)
	{attribute 'OPC.UA.DA' :='1'}
	popa_0082_ft_3122_b_low_delay_setpoint : INT;
	//Alarm active for HMI
	{attribute 'OPC.UA.DA' :='1'}
	popa_0082_ft_3122_b_low_active : BOOL;
	//Analog Alarm Setpoint
	{attribute 'OPC.UA.DA' :='1'}
	popa_0082_ft_3122_b_low_setpoint : REAL;
	//Alarm enable
	{attribute 'OPC.UA.DA' :='1'}
	popa_0082_ft_3122_b_low_enable: BOOL;
	
	//Alarm Priority setpoint
	{attribute 'OPC.UA.DA' :='1'}
	popa_0082_ft_3122_b_high_priority : INT;
	//Alarm delay setpoint(seconds)
	{attribute 'OPC.UA.DA' :='1'}
	popa_0082_ft_3122_b_high_delay_setpoint : INT;
	//Alarm active for HMI
	{attribute 'OPC.UA.DA' :='1'}
	popa_0082_ft_3122_b_high_active : BOOL;
	//Analog Alarm Setpoint
	{attribute 'OPC.UA.DA' :='1'}
	popa_0082_ft_3122_b_high_setpoint : REAL;
	//Alarm enable
	{attribute 'OPC.UA.DA' :='1'}
	popa_0082_ft_3122_b_high_enable: BOOL;
	
	//Alarm Priority setpoint
	{attribute 'OPC.UA.DA' :='1'}
	popa_0082_ft_3122_b_high_high_priority : INT;
	//Alarm delay setpoint(seconds)
	{attribute 'OPC.UA.DA' :='1'}
	popa_0082_ft_3122_b_high_high_delay_setpoint : INT;
	//Alarm active for HMI
	{attribute 'OPC.UA.DA' :='1'}
	popa_0082_ft_3122_b_high_high_active : BOOL;
	//Analog Alarm Setpoint
	{attribute 'OPC.UA.DA' :='1'}
	popa_0082_ft_3122_b_high_high_setpoint : REAL;
	//Alarm enable
	{attribute 'OPC.UA.DA' :='1'}
	popa_0082_ft_3122_b_high_high_enable: BOOL;
	
	
	//Raw Min value for analog input
	{attribute 'OPC.UA.DA' :='1'}
	popa_0082_ft_3122_b_raw_min : REAL :=0;
	//Raw max value for analog input
	{attribute 'OPC.UA.DA' :='1'}
	popa_0082_ft_3122_b_raw_max : REAL :=32767;
	//EU Min value for analog input
	{attribute 'OPC.UA.DA' :='1'}
	popa_0082_ft_3122_b_eu_min : REAL;
	//EU Max value for analog input
	{attribute 'OPC.UA.DA' :='1'}
	popa_0082_ft_3122_b_eu_max : REAL;
	//Filter factor value for analog input
	{attribute 'OPC.UA.DA' :='1'}
	popa_0082_ft_3122_b_filter_factor : REAL;
	//Scaled value for analog input
	{attribute 'OPC.UA.DA' :='1'}
	popa_0082_ft_3122_b_scaled_value : REAL;
	
	//---ft_3222-----------------------------------------------------------------------------------------------------------------------
	//Alarm Priority setpoint
	{attribute 'OPC.UA.DA' :='1'}
	popa_0082_ft_3222_b_low_low_priority : INT;
	//Alarm delay setpoint(seconds)
	{attribute 'OPC.UA.DA' :='1'}
	popa_0082_ft_3222_b_low_low_delay_setpoint : INT;
	//Alarm active for HMI
	{attribute 'OPC.UA.DA' :='1'}
	popa_0082_ft_3222_b_low_low_active : BOOL;
	//Analog Alarm Setpoint
	{attribute 'OPC.UA.DA' :='1'}
	popa_0082_ft_3222_b_low_low_setpoint : REAL;
	//Alarm enable
	{attribute 'OPC.UA.DA' :='1'}
	popa_0082_ft_3222_b_low_low_enable: BOOL;
	
	//Alarm Priority setpoint
	{attribute 'OPC.UA.DA' :='1'}
	popa_0082_ft_3222_b_low_priority : INT;
	//Alarm delay setpoint(seconds)
	{attribute 'OPC.UA.DA' :='1'}
	popa_0082_ft_3222_b_low_delay_setpoint : INT;
	//Alarm active for HMI
	{attribute 'OPC.UA.DA' :='1'}
	popa_0082_ft_3222_b_low_active : BOOL;
	//Analog Alarm Setpoint
	{attribute 'OPC.UA.DA' :='1'}
	popa_0082_ft_3222_b_low_setpoint : REAL;
	//Alarm enable
	{attribute 'OPC.UA.DA' :='1'}
	popa_0082_ft_3222_b_low_enable: BOOL;
	
	//Alarm Priority setpoint
	{attribute 'OPC.UA.DA' :='1'}
	popa_0082_ft_3222_b_high_priority : INT;
	//Alarm delay setpoint(seconds)
	{attribute 'OPC.UA.DA' :='1'}
	popa_0082_ft_3222_b_high_delay_setpoint : INT;
	//Alarm active for HMI
	{attribute 'OPC.UA.DA' :='1'}
	popa_0082_ft_3222_b_high_active : BOOL;
	//Analog Alarm Setpoint
	{attribute 'OPC.UA.DA' :='1'}
	popa_0082_ft_3222_b_high_setpoint : REAL;
	//Alarm enable
	{attribute 'OPC.UA.DA' :='1'}
	popa_0082_ft_3222_b_high_enable: BOOL;
	
	//Alarm Priority setpoint
	{attribute 'OPC.UA.DA' :='1'}
	popa_0082_ft_3222_b_high_high_priority : INT;
	//Alarm delay setpoint(seconds)
	{attribute 'OPC.UA.DA' :='1'}
	popa_0082_ft_3222_b_high_high_delay_setpoint : INT;
	//Alarm active for HMI
	{attribute 'OPC.UA.DA' :='1'}
	popa_0082_ft_3222_b_high_high_active : BOOL;
	//Analog Alarm Setpoint
	{attribute 'OPC.UA.DA' :='1'}
	popa_0082_ft_3222_b_high_high_setpoint : REAL;
	//Alarm enable
	{attribute 'OPC.UA.DA' :='1'}
	popa_0082_ft_3222_b_high_high_enable: BOOL;
	
	
	//Raw Min value for analog input
	{attribute 'OPC.UA.DA' :='1'}
	popa_0082_ft_3222_b_raw_min : REAL :=0;
	//Raw max value for analog input
	{attribute 'OPC.UA.DA' :='1'}
	popa_0082_ft_3222_b_raw_max : REAL :=32767;
	//EU Min value for analog input
	{attribute 'OPC.UA.DA' :='1'}
	popa_0082_ft_3222_b_eu_min : REAL;
	//EU Max value for analog input
	{attribute 'OPC.UA.DA' :='1'}
	popa_0082_ft_3222_b_eu_max : REAL;
	//Filter factor value for analog input
	{attribute 'OPC.UA.DA' :='1'}
	popa_0082_ft_3222_b_filter_factor : REAL;
	//Scaled value for analog input
	{attribute 'OPC.UA.DA' :='1'}
	popa_0082_ft_3222_b_scaled_value : REAL;
	
	//---ft_3322-----------------------------------------------------------------------------------------------------------------------
	//Alarm Priority setpoint
	{attribute 'OPC.UA.DA' :='1'}
	popa_0082_ft_3322_b_low_low_priority : INT;
	//Alarm delay setpoint(seconds)
	{attribute 'OPC.UA.DA' :='1'}
	popa_0082_ft_3322_b_low_low_delay_setpoint : INT;
	//Alarm active for HMI
	{attribute 'OPC.UA.DA' :='1'}
	popa_0082_ft_3322_b_low_low_active : BOOL;
	//Analog Alarm Setpoint
	{attribute 'OPC.UA.DA' :='1'}
	popa_0082_ft_3322_b_low_low_setpoint : REAL;
	//Alarm enable
	{attribute 'OPC.UA.DA' :='1'}
	popa_0082_ft_3322_b_low_low_enable: BOOL;
	
	//Alarm Priority setpoint
	{attribute 'OPC.UA.DA' :='1'}
	popa_0082_ft_3322_b_low_priority : INT;
	//Alarm delay setpoint(seconds)
	{attribute 'OPC.UA.DA' :='1'}
	popa_0082_ft_3322_b_low_delay_setpoint : INT;
	//Alarm active for HMI
	{attribute 'OPC.UA.DA' :='1'}
	popa_0082_ft_3322_b_low_active : BOOL;
	//Analog Alarm Setpoint
	{attribute 'OPC.UA.DA' :='1'}
	popa_0082_ft_3322_b_low_setpoint : REAL;
	//Alarm enable
	{attribute 'OPC.UA.DA' :='1'}
	popa_0082_ft_3322_b_low_enable: BOOL;
	
	//Alarm Priority setpoint
	{attribute 'OPC.UA.DA' :='1'}
	popa_0082_ft_3322_b_high_priority : INT;
	//Alarm delay setpoint(seconds)
	{attribute 'OPC.UA.DA' :='1'}
	popa_0082_ft_3322_b_high_delay_setpoint : INT;
	//Alarm active for HMI
	{attribute 'OPC.UA.DA' :='1'}
	popa_0082_ft_3322_b_high_active : BOOL;
	//Analog Alarm Setpoint
	{attribute 'OPC.UA.DA' :='1'}
	popa_0082_ft_3322_b_high_setpoint : REAL;
	//Alarm enable
	{attribute 'OPC.UA.DA' :='1'}
	popa_0082_ft_3322_b_high_enable: BOOL;
	
	//Alarm Priority setpoint
	{attribute 'OPC.UA.DA' :='1'}
	popa_0082_ft_3322_b_high_high_priority : INT;
	//Alarm delay setpoint(seconds)
	{attribute 'OPC.UA.DA' :='1'}
	popa_0082_ft_3322_b_high_high_delay_setpoint : INT;
	//Alarm active for HMI
	{attribute 'OPC.UA.DA' :='1'}
	popa_0082_ft_3322_b_high_high_active : BOOL;
	//Analog Alarm Setpoint
	{attribute 'OPC.UA.DA' :='1'}
	popa_0082_ft_3322_b_high_high_setpoint : REAL;
	//Alarm enable
	{attribute 'OPC.UA.DA' :='1'}
	popa_0082_ft_3322_b_high_high_enable: BOOL;
	
	
	//Raw Min value for analog input
	{attribute 'OPC.UA.DA' :='1'}
	popa_0082_ft_3322_b_raw_min : REAL :=0;
	//Raw max value for analog input
	{attribute 'OPC.UA.DA' :='1'}
	popa_0082_ft_3322_b_raw_max : REAL :=32767;
	//EU Min value for analog input
	{attribute 'OPC.UA.DA' :='1'}
	popa_0082_ft_3322_b_eu_min : REAL;
	//EU Max value for analog input
	{attribute 'OPC.UA.DA' :='1'}
	popa_0082_ft_3322_b_eu_max : REAL;
	//Filter factor value for analog input
	{attribute 'OPC.UA.DA' :='1'}
	popa_0082_ft_3322_b_filter_factor : REAL;
	//Scaled value for analog input
	{attribute 'OPC.UA.DA' :='1'}
	popa_0082_ft_3322_b_scaled_value : REAL;
	
	//---lt_3102-----------------------------------------------------------------------------------------------------------------------
	//Alarm Priority setpoint
	{attribute 'OPC.UA.DA' :='1'}
	popa_0082_lt_3102_b_low_low_priority : INT;
	//Alarm delay setpoint(seconds)
	{attribute 'OPC.UA.DA' :='1'}
	popa_0082_lt_3102_b_low_low_delay_setpoint : INT;
	//Alarm active for HMI
	{attribute 'OPC.UA.DA' :='1'}
	popa_0082_lt_3102_b_low_low_active : BOOL;
	//Analog Alarm Setpoint
	{attribute 'OPC.UA.DA' :='1'}
	popa_0082_lt_3102_b_low_low_setpoint : REAL;
	//Alarm enable
	{attribute 'OPC.UA.DA' :='1'}
	popa_0082_lt_3102_b_low_low_enable: BOOL;
	
	//Alarm Priority setpoint
	{attribute 'OPC.UA.DA' :='1'}
	popa_0082_lt_3102_b_low_priority : INT;
	//Alarm delay setpoint(seconds)
	{attribute 'OPC.UA.DA' :='1'}
	popa_0082_lt_3102_b_low_delay_setpoint : INT;
	//Alarm active for HMI
	{attribute 'OPC.UA.DA' :='1'}
	popa_0082_lt_3102_b_low_active : BOOL;
	//Analog Alarm Setpoint
	{attribute 'OPC.UA.DA' :='1'}
	popa_0082_lt_3102_b_low_setpoint : REAL;
	//Alarm enable
	{attribute 'OPC.UA.DA' :='1'}
	popa_0082_lt_3102_b_low_enable: BOOL;
	
	//Alarm Priority setpoint
	{attribute 'OPC.UA.DA' :='1'}
	popa_0082_lt_3102_b_high_priority : INT;
	//Alarm delay setpoint(seconds)
	{attribute 'OPC.UA.DA' :='1'}
	popa_0082_lt_3102_b_high_delay_setpoint : INT;
	//Alarm active for HMI
	{attribute 'OPC.UA.DA' :='1'}
	popa_0082_lt_3102_b_high_active : BOOL;
	//Analog Alarm Setpoint
	{attribute 'OPC.UA.DA' :='1'}
	popa_0082_lt_3102_b_high_setpoint : REAL;
	//Alarm enable
	{attribute 'OPC.UA.DA' :='1'}
	popa_0082_lt_3102_b_high_enable: BOOL;
	
	//Alarm Priority setpoint
	{attribute 'OPC.UA.DA' :='1'}
	popa_0082_lt_3102_b_high_high_priority : INT;
	//Alarm delay setpoint(seconds)
	{attribute 'OPC.UA.DA' :='1'}
	popa_0082_lt_3102_b_high_high_delay_setpoint : INT;
	//Alarm active for HMI
	{attribute 'OPC.UA.DA' :='1'}
	popa_0082_lt_3102_b_high_high_active : BOOL;
	//Analog Alarm Setpoint
	{attribute 'OPC.UA.DA' :='1'}
	popa_0082_lt_3102_b_high_high_setpoint : REAL;
	//Alarm enable
	{attribute 'OPC.UA.DA' :='1'}
	popa_0082_lt_3102_b_high_high_enable: BOOL;
	
	
	//Raw Min value for analog input
	{attribute 'OPC.UA.DA' :='1'}
	popa_0082_lt_3102_b_raw_min : REAL :=0;
	//Raw max value for analog input
	{attribute 'OPC.UA.DA' :='1'}
	popa_0082_lt_3102_b_raw_max : REAL :=32767;
	//EU Min value for analog input
	{attribute 'OPC.UA.DA' :='1'}
	popa_0082_lt_3102_b_eu_min : REAL;
	//EU Max value for analog input
	{attribute 'OPC.UA.DA' :='1'}
	popa_0082_lt_3102_b_eu_max : REAL;
	//Filter factor value for analog input
	{attribute 'OPC.UA.DA' :='1'}
	popa_0082_lt_3102_b_filter_factor : REAL;
	//Scaled value for analog input
	{attribute 'OPC.UA.DA' :='1'}
	popa_0082_lt_3102_b_scaled_value : REAL;
	
	//---lt_3202-----------------------------------------------------------------------------------------------------------------------
	//Alarm Priority setpoint
	{attribute 'OPC.UA.DA' :='1'}
	popa_0082_lt_3202_b_low_low_priority : INT;
	//Alarm delay setpoint(seconds)
	{attribute 'OPC.UA.DA' :='1'}
	popa_0082_lt_3202_b_low_low_delay_setpoint : INT;
	//Alarm active for HMI
	{attribute 'OPC.UA.DA' :='1'}
	popa_0082_lt_3202_b_low_low_active : BOOL;
	//Analog Alarm Setpoint
	{attribute 'OPC.UA.DA' :='1'}
	popa_0082_lt_3202_b_low_low_setpoint : REAL;
	//Alarm enable
	{attribute 'OPC.UA.DA' :='1'}
	popa_0082_lt_3202_b_low_low_enable: BOOL;
	
	//Alarm Priority setpoint
	{attribute 'OPC.UA.DA' :='1'}
	popa_0082_lt_3202_b_low_priority : INT;
	//Alarm delay setpoint(seconds)
	{attribute 'OPC.UA.DA' :='1'}
	popa_0082_lt_3202_b_low_delay_setpoint : INT;
	//Alarm active for HMI
	{attribute 'OPC.UA.DA' :='1'}
	popa_0082_lt_3202_b_low_active : BOOL;
	//Analog Alarm Setpoint
	{attribute 'OPC.UA.DA' :='1'}
	popa_0082_lt_3202_b_low_setpoint : REAL;
	//Alarm enable
	{attribute 'OPC.UA.DA' :='1'}
	popa_0082_lt_3202_b_low_enable: BOOL;
	
	//Alarm Priority setpoint
	{attribute 'OPC.UA.DA' :='1'}
	popa_0082_lt_3202_b_high_priority : INT;
	//Alarm delay setpoint(seconds)
	{attribute 'OPC.UA.DA' :='1'}
	popa_0082_lt_3202_b_high_delay_setpoint : INT;
	//Alarm active for HMI
	{attribute 'OPC.UA.DA' :='1'}
	popa_0082_lt_3202_b_high_active : BOOL;
	//Analog Alarm Setpoint
	{attribute 'OPC.UA.DA' :='1'}
	popa_0082_lt_3202_b_high_setpoint : REAL;
	//Alarm enable
	{attribute 'OPC.UA.DA' :='1'}
	popa_0082_lt_3202_b_high_enable: BOOL;
	
	//Alarm Priority setpoint
	{attribute 'OPC.UA.DA' :='1'}
	popa_0082_lt_3202_b_high_high_priority : INT;
	//Alarm delay setpoint(seconds)
	{attribute 'OPC.UA.DA' :='1'}
	popa_0082_lt_3202_b_high_high_delay_setpoint : INT;
	//Alarm active for HMI
	{attribute 'OPC.UA.DA' :='1'}
	popa_0082_lt_3202_b_high_high_active : BOOL;
	//Analog Alarm Setpoint
	{attribute 'OPC.UA.DA' :='1'}
	popa_0082_lt_3202_b_high_high_setpoint : REAL;
	//Alarm enable
	{attribute 'OPC.UA.DA' :='1'}
	popa_0082_lt_3202_b_high_high_enable: BOOL;
	
	
	//Raw Min value for analog input
	{attribute 'OPC.UA.DA' :='1'}
	popa_0082_lt_3202_b_raw_min : REAL :=0;
	//Raw max value for analog input
	{attribute 'OPC.UA.DA' :='1'}
	popa_0082_lt_3202_b_raw_max : REAL :=32767;
	//EU Min value for analog input
	{attribute 'OPC.UA.DA' :='1'}
	popa_0082_lt_3202_b_eu_min : REAL;
	//EU Max value for analog input
	{attribute 'OPC.UA.DA' :='1'}
	popa_0082_lt_3202_b_eu_max : REAL;
	//Filter factor value for analog input
	{attribute 'OPC.UA.DA' :='1'}
	popa_0082_lt_3202_b_filter_factor : REAL;
	//Scaled value for analog input
	{attribute 'OPC.UA.DA' :='1'}
	popa_0082_lt_3202_b_scaled_value : REAL;
	
	//---lt_3302-----------------------------------------------------------------------------------------------------------------------
	//Alarm Priority setpoint
	{attribute 'OPC.UA.DA' :='1'}
	popa_0082_lt_3302_b_low_low_priority : INT;
	//Alarm delay setpoint(seconds)
	{attribute 'OPC.UA.DA' :='1'}
	popa_0082_lt_3302_b_low_low_delay_setpoint : INT;
	//Alarm active for HMI
	{attribute 'OPC.UA.DA' :='1'}
	popa_0082_lt_3302_b_low_low_active : BOOL;
	//Analog Alarm Setpoint
	{attribute 'OPC.UA.DA' :='1'}
	popa_0082_lt_3302_b_low_low_setpoint : REAL;
	//Alarm enable
	{attribute 'OPC.UA.DA' :='1'}
	popa_0082_lt_3302_b_low_low_enable: BOOL;
	
	//Alarm Priority setpoint
	{attribute 'OPC.UA.DA' :='1'}
	popa_0082_lt_3302_b_low_priority : INT;
	//Alarm delay setpoint(seconds)
	{attribute 'OPC.UA.DA' :='1'}
	popa_0082_lt_3302_b_low_delay_setpoint : INT;
	//Alarm active for HMI
	{attribute 'OPC.UA.DA' :='1'}
	popa_0082_lt_3302_b_low_active : BOOL;
	//Analog Alarm Setpoint
	{attribute 'OPC.UA.DA' :='1'}
	popa_0082_lt_3302_b_low_setpoint : REAL;
	//Alarm enable
	{attribute 'OPC.UA.DA' :='1'}
	popa_0082_lt_3302_b_low_enable: BOOL;
	
	//Alarm Priority setpoint
	{attribute 'OPC.UA.DA' :='1'}
	popa_0082_lt_3302_b_high_priority : INT;
	//Alarm delay setpoint(seconds)
	{attribute 'OPC.UA.DA' :='1'}
	popa_0082_lt_3302_b_high_delay_setpoint : INT;
	//Alarm active for HMI
	{attribute 'OPC.UA.DA' :='1'}
	popa_0082_lt_3302_b_high_active : BOOL;
	//Analog Alarm Setpoint
	{attribute 'OPC.UA.DA' :='1'}
	popa_0082_lt_3302_b_high_setpoint : REAL;
	//Alarm enable
	{attribute 'OPC.UA.DA' :='1'}
	popa_0082_lt_3302_b_high_enable: BOOL;
	
	//Alarm Priority setpoint
	{attribute 'OPC.UA.DA' :='1'}
	popa_0082_lt_3302_b_high_high_priority : INT;
	//Alarm delay setpoint(seconds)
	{attribute 'OPC.UA.DA' :='1'}
	popa_0082_lt_3302_b_high_high_delay_setpoint : INT;
	//Alarm active for HMI
	{attribute 'OPC.UA.DA' :='1'}
	popa_0082_lt_3302_b_high_high_active : BOOL;
	//Analog Alarm Setpoint
	{attribute 'OPC.UA.DA' :='1'}
	popa_0082_lt_3302_b_high_high_setpoint : REAL;
	//Alarm enable
	{attribute 'OPC.UA.DA' :='1'}
	popa_0082_lt_3302_b_high_high_enable: BOOL;
	
	
	//Raw Min value for analog input
	{attribute 'OPC.UA.DA' :='1'}
	popa_0082_lt_3302_b_raw_min : REAL :=0;
	//Raw max value for analog input
	{attribute 'OPC.UA.DA' :='1'}
	popa_0082_lt_3302_b_raw_max : REAL :=32767;
	//EU Min value for analog input
	{attribute 'OPC.UA.DA' :='1'}
	popa_0082_lt_3302_b_eu_min : REAL;
	//EU Max value for analog input
	{attribute 'OPC.UA.DA' :='1'}
	popa_0082_lt_3302_b_eu_max : REAL;
	//Filter factor value for analog input
	{attribute 'OPC.UA.DA' :='1'}
	popa_0082_lt_3302_b_filter_factor : REAL;
	//Scaled value for analog input
	{attribute 'OPC.UA.DA' :='1'}
	popa_0082_lt_3302_b_scaled_value : REAL;
	
	//---lt_3153-----------------------------------------------------------------------------------------------------------------------
	//Alarm Priority setpoint
	{attribute 'OPC.UA.DA' :='1'}
	popa_0082_lt_3153_b_low_low_priority : INT;
	//Alarm delay setpoint(seconds)
	{attribute 'OPC.UA.DA' :='1'}
	popa_0082_lt_3153_b_low_low_delay_setpoint : INT;
	//Alarm active for HMI
	{attribute 'OPC.UA.DA' :='1'}
	popa_0082_lt_3153_b_low_low_active : BOOL;
	//Analog Alarm Setpoint
	{attribute 'OPC.UA.DA' :='1'}
	popa_0082_lt_3153_b_low_low_setpoint : REAL;
	//Alarm enable
	{attribute 'OPC.UA.DA' :='1'}
	popa_0082_lt_3153_b_low_low_enable: BOOL;
	
	//Alarm Priority setpoint
	{attribute 'OPC.UA.DA' :='1'}
	popa_0082_lt_3153_b_low_priority : INT;
	//Alarm delay setpoint(seconds)
	{attribute 'OPC.UA.DA' :='1'}
	popa_0082_lt_3153_b_low_delay_setpoint : INT;
	//Alarm active for HMI
	{attribute 'OPC.UA.DA' :='1'}
	popa_0082_lt_3153_b_low_active : BOOL;
	//Analog Alarm Setpoint
	{attribute 'OPC.UA.DA' :='1'}
	popa_0082_lt_3153_b_low_setpoint : REAL;
	//Alarm enable
	{attribute 'OPC.UA.DA' :='1'}
	popa_0082_lt_3153_b_low_enable: BOOL;
	
	//Alarm Priority setpoint
	{attribute 'OPC.UA.DA' :='1'}
	popa_0082_lt_3153_b_high_priority : INT;
	//Alarm delay setpoint(seconds)
	{attribute 'OPC.UA.DA' :='1'}
	popa_0082_lt_3153_b_high_delay_setpoint : INT;
	//Alarm active for HMI
	{attribute 'OPC.UA.DA' :='1'}
	popa_0082_lt_3153_b_high_active : BOOL;
	//Analog Alarm Setpoint
	{attribute 'OPC.UA.DA' :='1'}
	popa_0082_lt_3153_b_high_setpoint : REAL;
	//Alarm enable
	{attribute 'OPC.UA.DA' :='1'}
	popa_0082_lt_3153_b_high_enable: BOOL;
	
	//Alarm Priority setpoint
	{attribute 'OPC.UA.DA' :='1'}
	popa_0082_lt_3153_b_high_high_priority : INT;
	//Alarm delay setpoint(seconds)
	{attribute 'OPC.UA.DA' :='1'}
	popa_0082_lt_3153_b_high_high_delay_setpoint : INT;
	//Alarm active for HMI
	{attribute 'OPC.UA.DA' :='1'}
	popa_0082_lt_3153_b_high_high_active : BOOL;
	//Analog Alarm Setpoint
	{attribute 'OPC.UA.DA' :='1'}
	popa_0082_lt_3153_b_high_high_setpoint : REAL;
	//Alarm enable
	{attribute 'OPC.UA.DA' :='1'}
	popa_0082_lt_3153_b_high_high_enable: BOOL;
	
	
	//Raw Min value for analog input
	{attribute 'OPC.UA.DA' :='1'}
	popa_0082_lt_3153_b_raw_min : REAL :=0;
	//Raw max value for analog input
	{attribute 'OPC.UA.DA' :='1'}
	popa_0082_lt_3153_b_raw_max : REAL :=32767;
	//EU Min value for analog input
	{attribute 'OPC.UA.DA' :='1'}
	popa_0082_lt_3153_b_eu_min : REAL;
	//EU Max value for analog input
	{attribute 'OPC.UA.DA' :='1'}
	popa_0082_lt_3153_b_eu_max : REAL;
	//Filter factor value for analog input
	{attribute 'OPC.UA.DA' :='1'}
	popa_0082_lt_3153_b_filter_factor : REAL;
	//Scaled value for analog input
	{attribute 'OPC.UA.DA' :='1'}
	popa_0082_lt_3153_b_scaled_value : REAL;
	
	//---lt_3253-----------------------------------------------------------------------------------------------------------------------
	//Alarm Priority setpoint
	{attribute 'OPC.UA.DA' :='1'}
	popa_0082_lt_3253_b_low_low_priority : INT;
	//Alarm delay setpoint(seconds)
	{attribute 'OPC.UA.DA' :='1'}
	popa_0082_lt_3253_b_low_low_delay_setpoint : INT;
	//Alarm active for HMI
	{attribute 'OPC.UA.DA' :='1'}
	popa_0082_lt_3253_b_low_low_active : BOOL;
	//Analog Alarm Setpoint
	{attribute 'OPC.UA.DA' :='1'}
	popa_0082_lt_3253_b_low_low_setpoint : REAL;
	//Alarm enable
	{attribute 'OPC.UA.DA' :='1'}
	popa_0082_lt_3253_b_low_low_enable: BOOL;
	
	//Alarm Priority setpoint
	{attribute 'OPC.UA.DA' :='1'}
	popa_0082_lt_3253_b_low_priority : INT;
	//Alarm delay setpoint(seconds)
	{attribute 'OPC.UA.DA' :='1'}
	popa_0082_lt_3253_b_low_delay_setpoint : INT;
	//Alarm active for HMI
	{attribute 'OPC.UA.DA' :='1'}
	popa_0082_lt_3253_b_low_active : BOOL;
	//Analog Alarm Setpoint
	{attribute 'OPC.UA.DA' :='1'}
	popa_0082_lt_3253_b_low_setpoint : REAL;
	//Alarm enable
	{attribute 'OPC.UA.DA' :='1'}
	popa_0082_lt_3253_b_low_enable: BOOL;
	
	//Alarm Priority setpoint
	{attribute 'OPC.UA.DA' :='1'}
	popa_0082_lt_3253_b_high_priority : INT;
	//Alarm delay setpoint(seconds)
	{attribute 'OPC.UA.DA' :='1'}
	popa_0082_lt_3253_b_high_delay_setpoint : INT;
	//Alarm active for HMI
	{attribute 'OPC.UA.DA' :='1'}
	popa_0082_lt_3253_b_high_active : BOOL;
	//Analog Alarm Setpoint
	{attribute 'OPC.UA.DA' :='1'}
	popa_0082_lt_3253_b_high_setpoint : REAL;
	//Alarm enable
	{attribute 'OPC.UA.DA' :='1'}
	popa_0082_lt_3253_b_high_enable: BOOL;
	
	//Alarm Priority setpoint
	{attribute 'OPC.UA.DA' :='1'}
	popa_0082_lt_3253_b_high_high_priority : INT;
	//Alarm delay setpoint(seconds)
	{attribute 'OPC.UA.DA' :='1'}
	popa_0082_lt_3253_b_high_high_delay_setpoint : INT;
	//Alarm active for HMI
	{attribute 'OPC.UA.DA' :='1'}
	popa_0082_lt_3253_b_high_high_active : BOOL;
	//Analog Alarm Setpoint
	{attribute 'OPC.UA.DA' :='1'}
	popa_0082_lt_3253_b_high_high_setpoint : REAL;
	//Alarm enable
	{attribute 'OPC.UA.DA' :='1'}
	popa_0082_lt_3253_b_high_high_enable: BOOL;
	
	
	//Raw Min value for analog input
	{attribute 'OPC.UA.DA' :='1'}
	popa_0082_lt_3253_b_raw_min : REAL :=0;
	//Raw max value for analog input
	{attribute 'OPC.UA.DA' :='1'}
	popa_0082_lt_3253_b_raw_max : REAL :=32767;
	//EU Min value for analog input
	{attribute 'OPC.UA.DA' :='1'}
	popa_0082_lt_3253_b_eu_min : REAL;
	//EU Max value for analog input
	{attribute 'OPC.UA.DA' :='1'}
	popa_0082_lt_3253_b_eu_max : REAL;
	//Filter factor value for analog input
	{attribute 'OPC.UA.DA' :='1'}
	popa_0082_lt_3253_b_filter_factor : REAL;
	//Scaled value for analog input
	{attribute 'OPC.UA.DA' :='1'}
	popa_0082_lt_3253_b_scaled_value : REAL;
	
	//---lt_3353-----------------------------------------------------------------------------------------------------------------------
	//Alarm Priority setpoint
	{attribute 'OPC.UA.DA' :='1'}
	popa_0082_lt_3353_b_low_low_priority : INT;
	//Alarm delay setpoint(seconds)
	{attribute 'OPC.UA.DA' :='1'}
	popa_0082_lt_3353_b_low_low_delay_setpoint : INT;
	//Alarm active for HMI
	{attribute 'OPC.UA.DA' :='1'}
	popa_0082_lt_3353_b_low_low_active : BOOL;
	//Analog Alarm Setpoint
	{attribute 'OPC.UA.DA' :='1'}
	popa_0082_lt_3353_b_low_low_setpoint : REAL;
	//Alarm enable
	{attribute 'OPC.UA.DA' :='1'}
	popa_0082_lt_3353_b_low_low_enable: BOOL;
	
	//Alarm Priority setpoint
	{attribute 'OPC.UA.DA' :='1'}
	popa_0082_lt_3353_b_low_priority : INT;
	//Alarm delay setpoint(seconds)
	{attribute 'OPC.UA.DA' :='1'}
	popa_0082_lt_3353_b_low_delay_setpoint : INT;
	//Alarm active for HMI
	{attribute 'OPC.UA.DA' :='1'}
	popa_0082_lt_3353_b_low_active : BOOL;
	//Analog Alarm Setpoint
	{attribute 'OPC.UA.DA' :='1'}
	popa_0082_lt_3353_b_low_setpoint : REAL;
	//Alarm enable
	{attribute 'OPC.UA.DA' :='1'}
	popa_0082_lt_3353_b_low_enable: BOOL;
	
	//Alarm Priority setpoint
	{attribute 'OPC.UA.DA' :='1'}
	popa_0082_lt_3353_b_high_priority : INT;
	//Alarm delay setpoint(seconds)
	{attribute 'OPC.UA.DA' :='1'}
	popa_0082_lt_3353_b_high_delay_setpoint : INT;
	//Alarm active for HMI
	{attribute 'OPC.UA.DA' :='1'}
	popa_0082_lt_3353_b_high_active : BOOL;
	//Analog Alarm Setpoint
	{attribute 'OPC.UA.DA' :='1'}
	popa_0082_lt_3353_b_high_setpoint : REAL;
	//Alarm enable
	{attribute 'OPC.UA.DA' :='1'}
	popa_0082_lt_3353_b_high_enable: BOOL;
	
	//Alarm Priority setpoint
	{attribute 'OPC.UA.DA' :='1'}
	popa_0082_lt_3353_b_high_high_priority : INT;
	//Alarm delay setpoint(seconds)
	{attribute 'OPC.UA.DA' :='1'}
	popa_0082_lt_3353_b_high_high_delay_setpoint : INT;
	//Alarm active for HMI
	{attribute 'OPC.UA.DA' :='1'}
	popa_0082_lt_3353_b_high_high_active : BOOL;
	//Analog Alarm Setpoint
	{attribute 'OPC.UA.DA' :='1'}
	popa_0082_lt_3353_b_high_high_setpoint : REAL;
	//Alarm enable
	{attribute 'OPC.UA.DA' :='1'}
	popa_0082_lt_3353_b_high_high_enable: BOOL;
	
	
	//Raw Min value for analog input
	{attribute 'OPC.UA.DA' :='1'}
	popa_0082_lt_3353_b_raw_min : REAL :=0;
	//Raw max value for analog input
	{attribute 'OPC.UA.DA' :='1'}
	popa_0082_lt_3353_b_raw_max : REAL :=32767;
	//EU Min value for analog input
	{attribute 'OPC.UA.DA' :='1'}
	popa_0082_lt_3353_b_eu_min : REAL;
	//EU Max value for analog input
	{attribute 'OPC.UA.DA' :='1'}
	popa_0082_lt_3353_b_eu_max : REAL;
	//Filter factor value for analog input
	{attribute 'OPC.UA.DA' :='1'}
	popa_0082_lt_3353_b_filter_factor : REAL;
	//Scaled value for analog input
	{attribute 'OPC.UA.DA' :='1'}
	popa_0082_lt_3353_b_scaled_value : REAL;
	
	//---lt_3402-----------------------------------------------------------------------------------------------------------------------
	//Alarm Priority setpoint
	{attribute 'OPC.UA.DA' :='1'}
	popa_0092_lt_3402_b_low_low_priority : INT;
	//Alarm delay setpoint(seconds)
	{attribute 'OPC.UA.DA' :='1'}
	popa_0092_lt_3402_b_low_low_delay_setpoint : INT;
	//Alarm active for HMI
	{attribute 'OPC.UA.DA' :='1'}
	popa_0092_lt_3402_b_low_low_active : BOOL;
	//Analog Alarm Setpoint
	{attribute 'OPC.UA.DA' :='1'}
	popa_0092_lt_3402_b_low_low_setpoint : REAL;
	//Alarm enable
	{attribute 'OPC.UA.DA' :='1'}
	popa_0092_lt_3402_b_low_low_enable: BOOL;
	
	//Alarm Priority setpoint
	{attribute 'OPC.UA.DA' :='1'}
	popa_0092_lt_3402_b_low_priority : INT;
	//Alarm delay setpoint(seconds)
	{attribute 'OPC.UA.DA' :='1'}
	popa_0092_lt_3402_b_low_delay_setpoint : INT;
	//Alarm active for HMI
	{attribute 'OPC.UA.DA' :='1'}
	popa_0092_lt_3402_b_low_active : BOOL;
	//Analog Alarm Setpoint
	{attribute 'OPC.UA.DA' :='1'}
	popa_0092_lt_3402_b_low_setpoint : REAL;
	//Alarm enable
	{attribute 'OPC.UA.DA' :='1'}
	popa_0092_lt_3402_b_low_enable: BOOL;
	
	//Alarm Priority setpoint
	{attribute 'OPC.UA.DA' :='1'}
	popa_0092_lt_3402_b_high_priority : INT;
	//Alarm delay setpoint(seconds)
	{attribute 'OPC.UA.DA' :='1'}
	popa_0092_lt_3402_b_high_delay_setpoint : INT;
	//Alarm active for HMI
	{attribute 'OPC.UA.DA' :='1'}
	popa_0092_lt_3402_b_high_active : BOOL;
	//Analog Alarm Setpoint
	{attribute 'OPC.UA.DA' :='1'}
	popa_0092_lt_3402_b_high_setpoint : REAL;
	//Alarm enable
	{attribute 'OPC.UA.DA' :='1'}
	popa_0092_lt_3402_b_high_enable: BOOL;
	
	//Alarm Priority setpoint
	{attribute 'OPC.UA.DA' :='1'}
	popa_0092_lt_3402_b_high_high_priority : INT;
	//Alarm delay setpoint(seconds)
	{attribute 'OPC.UA.DA' :='1'}
	popa_0092_lt_3402_b_high_high_delay_setpoint : INT;
	//Alarm active for HMI
	{attribute 'OPC.UA.DA' :='1'}
	popa_0092_lt_3402_b_high_high_active : BOOL;
	//Analog Alarm Setpoint
	{attribute 'OPC.UA.DA' :='1'}
	popa_0092_lt_3402_b_high_high_setpoint : REAL;
	//Alarm enable
	{attribute 'OPC.UA.DA' :='1'}
	popa_0092_lt_3402_b_high_high_enable: BOOL;
	
	
	//Raw Min value for analog input
	{attribute 'OPC.UA.DA' :='1'}
	popa_0092_lt_3402_b_raw_min : REAL :=0;
	//Raw max value for analog input
	{attribute 'OPC.UA.DA' :='1'}
	popa_0092_lt_3402_b_raw_max : REAL :=32767;
	//EU Min value for analog input
	{attribute 'OPC.UA.DA' :='1'}
	popa_0092_lt_3402_b_eu_min : REAL;
	//EU Max value for analog input
	{attribute 'OPC.UA.DA' :='1'}
	popa_0092_lt_3402_b_eu_max : REAL;
	//Filter factor value for analog input
	{attribute 'OPC.UA.DA' :='1'}
	popa_0092_lt_3402_b_filter_factor : REAL;
	//Scaled value for analog input
	{attribute 'OPC.UA.DA' :='1'}
	popa_0092_lt_3402_b_scaled_value : REAL;
	
	
	//---pt_3119-----------------------------------------------------------------------------------------------------------------------
	//Alarm Priority setpoint
	{attribute 'OPC.UA.DA' :='1'}
	popa_0082_pt_3119_b_low_low_priority : INT;
	//Alarm delay setpoint(seconds)
	{attribute 'OPC.UA.DA' :='1'}
	popa_0082_pt_3119_b_low_low_delay_setpoint : INT;
	//Alarm active for HMI
	{attribute 'OPC.UA.DA' :='1'}
	popa_0082_pt_3119_b_low_low_active : BOOL;
	//Analog Alarm Setpoint
	{attribute 'OPC.UA.DA' :='1'}
	popa_0082_pt_3119_b_low_low_setpoint : REAL;
	//Alarm enable
	{attribute 'OPC.UA.DA' :='1'}
	popa_0082_pt_3119_b_low_low_enable: BOOL;
	
